                   "Technology".Substage := 116; //процесс прогрева
               ELSE
                   "HMI".INDICATION_TIME_1 := 255;
                   "HMI".INDICATION_TIME_2 := 255;
                   "Technology".Substage := 0; //неизвестно
           END_CASE;
       8:  //работа
           CASE "Technology".Regim_run_step OF
               0:
                   IF NOT "Protections_BLOCK".Not_flame_burner THEN
                       "HMI".LTIME_converter_IN := "Timer_RUN_temp_DB".ET;
                       "HMI".INDICATION_TIME_1 := DINT_TO_USINT("HMI".LTIME_converter_day);
                       "HMI".INDICATION_TIME_2 := INT_TO_USINT("HMI".LTIME_converter_hour);
                   ELSE    //если имеется блокировка защиты по погасанию пламени горелки
                       "HMI".TIME_converter_IN := "TON_protection_13_DB".PT - "TON_protection_13_DB".ET;
                       "HMI".INDICATION_TIME_1 := INT_TO_USINT("HMI".TIME_converter_minute);
                       "HMI".INDICATION_TIME_2 := INT_TO_USINT("HMI".TIME_converter_second);
                   END_IF;
                   "Technology".Substage := 117; //процесс работы 
               ELSE
                   "HMI".INDICATION_TIME_1 := 255;
                   "HMI".INDICATION_TIME_2 := 255;
                   "Technology".Substage := 0; //неизвестно
           END_CASE;
       9:  //экстренный останов
           "HMI".INDICATION_TIME_1 := 255;
           "HMI".INDICATION_TIME_2 := 255;
           CASE "Technology".Regim_emergency_stop_step OF
               0:
                   IF NOT "Message".EMERGENCY_STOP_not_initial_state THEN
                       "Technology".Substage := 120; //отключение всего 
                   ELSE
                       "Technology".Substage := 121; //устройства не переведены в исходное состояние
                   END_IF;
               ELSE
                   "Technology".Substage := 0; //неизвестно
           END_CASE;
       10: //аварийный останов
           "HMI".INDICATION_TIME_1 := 255;
           "HMI".INDICATION_TIME_2 := 255;
           CASE "Technology".Regim_alarm_stop_step OF
               0:
                   IF NOT "Message".ALARM_STOP_not_initial_state_gas THEN
                       "Technology".Substage := 122; //перевод всех газовых клапанов в исходное состояние
                   ELSE
                       "Technology".Substage := 123; //газовые клапана не переведены в исходное состояние
                   END_IF;
               ELSE
                   "Technology".Substage := 0; //неизвестно
           END_CASE;
       11: //плановый останов
           "HMI".INDICATION_TIME_1 := 255;
           "HMI".INDICATION_TIME_2 := 255;
           CASE "Technology".Regim_plan_stop_step OF
               0:
                   "Technology".Substage := 130; //вывод ЗРГ на значение минимальной мощности
               1:
                   "Technology".Substage := 131; //вывод ЗРГ на значение минимальной мощности
               2:
                   IF NOT "Message".PLAN_STOP_not_initial_state_gas THEN
                       "Technology".Substage := 132; //перевод газовых клапанов в исходное состояние, регуляторов разряжения и вентиляции на вентиляционные параметры
                   ELSE
                       "Technology".Substage := 133; //газовые клапана не переведены в исходное состояние
                   END_IF;
               3:
                   "Technology".Substage := 134; //перевод регуляторов разряжения и вентиляции на вентиляционные параметры
               ELSE
                   "Technology".Substage := 0; //неизвестно
           END_CASE;
       12: //постостановочная опрессовка
           "HMI".INDICATION_TIME_1 := 255;
           "HMI".INDICATION_TIME_2 := 255;
           CASE "Technology".Regim_stop_press_step OF
               0:
                   "Technology".Substage := 140; //анализ разрешения проведения постостановочной опрессовки
               1:
                   "Technology".Substage := 141; //контроль положения исполнительных механизмов по газу
               2:
                   "Technology".Substage := 142; //контроль min P
               3:
                   "Technology".Substage := 143; //контроль max P
               4:
                   "Technology".Substage := 144; //закрываем КБ
               5:
                   "Technology".Substage := 145; //контроль отсутствия давления газа м/у ПЗК
               6:
                   "Technology".Substage := 146; //открываем КО
               7:
                   "Technology".Substage := 147; //контроль достижения давления газа м/у ПЗК
               8:
                   "Technology".Substage := 148; //закрываем КО
               9:
                   "Technology".Substage := 149; //открываем КБ
               10:
                   "Technology".Substage := 150; //определение успешности постостановочной опрессовки
               11:
                   IF "Message".STOP_PRESS_PZK1_or_KO_untight THEN
                       "Technology".Substage := 151; //постостановочная опрессовка не прошла. ПЗК1 или КО негерметичен
                   END_IF;
                   IF "Message".STOP_PRESS_PZK2_or_KB_untight THEN
                       "Technology".Substage := 152; //постостановочная опрессовка не прошла. ПЗК2 или КБ негерметичен
                   END_IF;
                   IF "Message".STOP_PRESS_P_before_BG_min THEN
                       "Technology".Substage := 153; //постостановочная опрессовка не прошла. Низкое давление до БГ
                   END_IF;
                   IF "Message".STOP_PRESS_success THEN
                       "Technology".Substage := 154; //постостановочная опрессовка успешно проведена
                   END_IF;
               ELSE
                   "Technology".Substage := 0; //неизвестно
           END_CASE;
       13: //укороченная вентиляция
           CASE "Technology".Regim_short_ventilation_step OF
               0:
                   "HMI".INDICATION_TIME_1 := 255;
                   "HMI".INDICATION_TIME_2 := 255;
                   "Technology".Substage := 160; //анализ необходимости проведения укороченной вентиляции
               1:
                   "HMI".INDICATION_TIME_1 := 255;
                   "HMI".INDICATION_TIME_2 := 255;
                   "Technology".Substage := 161; //переход на поддержание вентиляционного значения разрежения
               2:
                   "HMI".INDICATION_TIME_1 := 255;
                   "HMI".INDICATION_TIME_2 := 255;
                   "Technology".Substage := 162; //переход на поддержание вентиляционного значения разрежения
               3:
                   "HMI".INDICATION_TIME_1 := 255;
                   "HMI".INDICATION_TIME_2 := 255;
                   "Technology".Substage := 163; //переход на поддержание вентиляционного значения давления воздуха
               4:
                   "HMI".TIME_converter_IN := "Timer_SHORT_VENTILATION_temp_DB".PT - "Timer_SHORT_VENTILATION_temp_DB".ET;
                   "HMI".INDICATION_TIME_1 := INT_TO_USINT("HMI".TIME_converter_minute);
                   "HMI".INDICATION_TIME_2 := INT_TO_USINT("HMI".TIME_converter_second);
                   "Technology".Substage := 164; //процесс вентиляции
               5:
                   "HMI".INDICATION_TIME_1 := 255;
                   "HMI".INDICATION_TIME_2 := 255;
                   "Technology".Substage := 165; //переход на поддержание розжигового значения разрежения
               6:
                   "HMI".INDICATION_TIME_1 := 255;
                   "HMI".INDICATION_TIME_2 := 255;
                   "Technology".Substage := 166; //переход на поддержание розжигового значения разрежения
               7:
                   "HMI".INDICATION_TIME_1 := 255;
                   "HMI".INDICATION_TIME_2 := 255;
                   "Technology".Substage := 167; //переход на поддержание розжигового значения давления воздуха
               ELSE
                   "HMI".INDICATION_TIME_1 := 255;
                   "HMI".INDICATION_TIME_2 := 255;
                   "Technology".Substage := 0; //неизвестно
           END_CASE;
       ELSE
           "Technology".Substage := 0; //неизвестно
   END_CASE;

   "TIME_converter_DB"(IN := "HMI".TIME_converter_IN,
                       Minute => "HMI".TIME_converter_minute,
                       Second => "HMI".TIME_converter_second);

   "LTIME_converter_DB"(IN := "HMI".LTIME_converter_IN,
                        Day=>"HMI".LTIME_converter_day,
                        Hour=>"HMI".LTIME_converter_hour);
END_FUNCTION

FUNCTION "Protection" : Void   // FC9, SCL
{ S7_Optimized_Access := 'TRUE' }
VERSION : 0.1
BEGIN
   (*Принудительный сброс блокировок защит*)
   (*Невоспламенение или погасание факела горелки котла*)
   "TON_protection_13_DB".TON(IN :="Protections_BLOCK".Not_flame_burner,
   PT := T#5m,
   Q => "Timer".protection_13_Q);
   IF "Timer".protection_13_Q THEN
       "Protections_BLOCK".Not_flame_burner := FALSE;
   END_IF;

   (*формирование обобщенного признака сработки защиты*)
   IF "Protections".P_gas_before_BG_max OR
       "Protections".P_gas_before_BG_min OR
       "Protections".P_gas_before_burner_min OR
       "Protections".P_gas_before_burner_max OR
       "Protections".DS_off OR
       "Protections".DV_off OR
       "Protections".dP_in_furnance_min OR
       "Protections".P_air_before_burner_min OR
       "Protections".L_water_min OR
       "Protections".L_water_max OR
       "Protections".P_steam_max OR
       "Protections".Not_flame_burner OR
       "Protections".Alarm_stop_HMI OR
       "Protections".Alarm_stop_SCADA THEN
       "Protections".Global := TRUE;
   ELSE
       "Protections".Global := FALSE;
   END_IF;
END_FUNCTION

FUNCTION "Regim_map" : Void   // FC10, SCL
{ S7_Optimized_Access := 'TRUE' }
VERSION : 0.1
BEGIN
   (*Защита от неправильного ввода параметров режимной карты*)
   IF "RegMap".P_gaz_2 < "RegMap".P_gaz_1 THEN
       "RegMap".P_gaz_2 := "RegMap".P_gaz_1+0.1;
   END_IF;
   IF "RegMap".P_gaz_3 < "RegMap".P_gaz_2 THEN
       "RegMap".P_gaz_3 := "RegMap".P_gaz_2+0.1;
   END_IF;
   IF "RegMap".P_gaz_4 < "RegMap".P_gaz_3 THEN
       "RegMap".P_gaz_4 := "RegMap".P_gaz_3+0.1;
   END_IF;
   IF "RegMap".P_gaz_5 < "RegMap".P_gaz_4 THEN
       "RegMap".P_gaz_5 := "RegMap".P_gaz_4+0.1;
   END_IF;
   IF "RegMap".P_gaz_6 < "RegMap".P_gaz_5 THEN
       "RegMap".P_gaz_6 := "RegMap".P_gaz_5+0.1;
   END_IF;
   IF "RegMap".P_gaz_7 < "RegMap".P_gaz_6 THEN
       "RegMap".P_gaz_7 := "RegMap".P_gaz_6+0.1;
   END_IF;
   IF "RegMap".P_gaz_8 < "RegMap".P_gaz_7 THEN
       "RegMap".P_gaz_8 := "RegMap".P_gaz_7+0.1;
   END_IF;

   (*НАСТРОЙКА РЕЖИМНОЙ КАРТЫ*)
   (*давление воздуха*)
   "Polyline_P_air_DB"();

   "Polyline_P_air_DB".Input := "P_gas_before_burner".Value;

   "Polyline_P_air_DB".UserData.Point[1].x := "RegMap".P_gaz_1;
   "Polyline_P_air_DB".UserData.Point[2].x := "RegMap".P_gaz_2;
   "Polyline_P_air_DB".UserData.Point[3].x := "RegMap".P_gaz_3;
   "Polyline_P_air_DB".UserData.Point[4].x := "RegMap".P_gaz_4;
   "Polyline_P_air_DB".UserData.Point[5].x := "RegMap".P_gaz_5;
   "Polyline_P_air_DB".UserData.Point[6].x := "RegMap".P_gaz_6;
   "Polyline_P_air_DB".UserData.Point[7].x := "RegMap".P_gaz_7;
   "Polyline_P_air_DB".UserData.Point[8].x := "RegMap".P_gaz_8;

   "Polyline_P_air_DB".UserData.Point[1].y := "RegMap".P_air_1;
   "Polyline_P_air_DB".UserData.Point[2].y := "RegMap".P_air_2;
   "Polyline_P_air_DB".UserData.Point[3].y := "RegMap".P_air_3;
   "Polyline_P_air_DB".UserData.Point[4].y := "RegMap".P_air_4;
   "Polyline_P_air_DB".UserData.Point[5].y := "RegMap".P_air_5;
   "Polyline_P_air_DB".UserData.Point[6].y := "RegMap".P_air_6;
   "Polyline_P_air_DB".UserData.Point[7].y := "RegMap".P_air_7;
   "Polyline_P_air_DB".UserData.Point[8].y := "RegMap".P_air_8;

   (*разряжение*)
   "Polyline_dP_DB"();

   "Polyline_dP_DB".Input := "P_gas_before_burner".Value;

   "Polyline_dP_DB".UserData.Point[1].x := "RegMap".P_gaz_1;
   "Polyline_dP_DB".UserData.Point[2].x := "RegMap".P_gaz_2;
   "Polyline_dP_DB".UserData.Point[3].x := "RegMap".P_gaz_3;
   "Polyline_dP_DB".UserData.Point[4].x := "RegMap".P_gaz_4;
   "Polyline_dP_DB".UserData.Point[5].x := "RegMap".P_gaz_5;
   "Polyline_dP_DB".UserData.Point[6].x := "RegMap".P_gaz_6;
   "Polyline_dP_DB".UserData.Point[7].x := "RegMap".P_gaz_7;
   "Polyline_dP_DB".UserData.Point[8].x := "RegMap".P_gaz_8;

   "Polyline_dP_DB".UserData.Point[1].y := "RegMap".dP_furnace_1;
   "Polyline_dP_DB".UserData.Point[2].y := "RegMap".dP_furnace_2;
   "Polyline_dP_DB".UserData.Point[3].y := "RegMap".dP_furnace_3;
   "Polyline_dP_DB".UserData.Point[4].y := "RegMap".dP_furnace_4;
   "Polyline_dP_DB".UserData.Point[5].y := "RegMap".dP_furnace_5;
   "Polyline_dP_DB".UserData.Point[6].y := "RegMap".dP_furnace_6;
   "Polyline_dP_DB".UserData.Point[7].y := "RegMap".dP_furnace_7;
   "Polyline_dP_DB".UserData.Point[8].y := "RegMap".dP_furnace_8;

   (*Режимная карта. Применить. Для журнала событий*)
   IF "RegMap".Apply THEN
       "HMI".RegMap_Apply_Log := TRUE;
   END_IF;

   IF "Syst".First_scan_reg_map THEN
       "RegMap".Apply := TRUE;
       "Syst".First_scan_reg_map := FALSE;
   END_IF;

   //применить новые значения
   "Polyline_P_air_DB".Validate := "RegMap".Apply;
   "Polyline_dP_DB".Validate := "RegMap".Apply;
   IF "RegMap".Apply THEN
       "RegMap".Apply := FALSE;
   END_IF;

   //значение расчетных параметров
   "RegMap".P_air_regim_map := "Polyline_P_air_DB".Output;
   "RegMap".dP_furnace_regim_map := "Polyline_dP_DB".Output;

   //индикация ошибки
   "RegMap".Error := "Polyline_P_air_DB".Error OR "Polyline_dP_DB".Error;

   //сброс
   "Polyline_P_air_DB".Reset := "RegMap".Reset;
   "Polyline_dP_DB".Reset := "RegMap".Reset;
   IF "RegMap".Reset THEN
       "RegMap".Reset := FALSE;
   END_IF;
END_FUNCTION

FUNCTION "Log" : Void   // FC11, SCL
{ S7_Optimized_Access := 'TRUE' }
VERSION : 0.1
BEGIN
   (*Нажатие кнопок для журнала событий*)
   (*Кнопка ВЕНТИЛЯЦИЯ на панели оператора для журнала событий*)
   IF "HMI".Btn_Ventilation_HMI THEN
       "HMI".Btn_Ventilation_HMI_Log := TRUE;
   END_IF;
   (*Кнопка ВЕНТИЛЯЦИЯ на SCADA для журнала событий*)
   IF "HMI".Btn_Ventilation_SCADA THEN
       "HMI".Btn_Ventilation_SCADA_Log := TRUE;
   END_IF;
   (*Кнопка ВЕНТИЛЯЦИЯ на ШАУ для журнала событий*)
   IF "Btn_Ventilation".Value THEN
       "HMI".Btn_Ventilation_ShAU_Log := TRUE;
   END_IF;
   (*Кнопка РОЗЖИГ на панели оператора для журнала событий*)
   IF "HMI".Btn_Ignition_HMI THEN
       "HMI".Btn_Ignition_HMI_Log := TRUE;
   END_IF;
   (*Кнопка РОЗЖИГ на SCADA для журнала событий*)
   IF "HMI".Btn_Ignition_SCADA THEN
       "HMI".Btn_Ignition_SCADA_Log := TRUE;
   END_IF;
   (*Кнопка РОЗЖИГ на ШАУ для журнала событий*)
   IF "Btn_Ignition".Value THEN
       "HMI".Btn_Ignition_ShAU_Log := TRUE;
   END_IF;
   (*Кнопка НОРМАЛЬНЫЙ ОСТАНОВ на панели оператора для журнала событий*)
   IF "HMI".Btn_normal_stop_HMI THEN
       "HMI".Btn_normal_stop_HMI_Log := TRUE;
   END_IF;
   (*Кнопка НОРМАЛЬНЫЙ ОСТАНОВ на SCADA для журнала событий*)
   IF "HMI".Btn_normal_stop_SCADA THEN
       "HMI".Btn_normal_stop_SCADA_Log := TRUE;
   END_IF;
   (*Кнопка АВАРИЙНЫЙ ОСТАНОВ на панели оператора для журнала событий*)
   IF "HMI".Btn_alarm_stop_HMI THEN
       "HMI".Btn_alarm_stop_HMI_Log := TRUE;
   END_IF;
   (*Кнопка АВАРИЙНЫЙ ОСТАНОВ на SCADA для журнала событий*)
   IF "HMI".Btn_alarm_stop_SCADA THEN
       "HMI".Btn_alarm_stop_SCADA_Log := TRUE;
   END_IF;
   (*Кнопка ЭКСТРЕННЫЙ ОСТАНОВ на ШАУ для журнала событий*)
   IF "Btn_STOP".Value THEN
       "HMI".Btn_emergency_stop_ShAU_Log := TRUE;
   END_IF;
   (*Кнопка ТЕСТОВАЯ ОПРЕССОВКА на панели оператора для журнала событий*)
   IF "HMI".Btn_test_press_HMI THEN
       "HMI".Btn_test_press_HMI_Log := TRUE;
   END_IF;
   (*Кнопка ТЕСТОВЫЙ РОЗЖИГ на панели оператора для журнала событий*)
   IF "HMI".Btn_test_ignition_HMI THEN
       "HMI".Btn_test_ignition_HMI_Log := TRUE;
   END_IF;
   (*Кнопка Ручной РОЗЖИГ на панели оператора для журнала событий*)
   IF "HMI".Btn_manual_ignition_HMI THEN
       "HMI".Btn_manual_ignition_HMI_Log := TRUE;
   END_IF;
   (*Кнопка СБРОС ЗВУКА на панели оператора для журнала событий*)
   IF "HMI".Btn_reset_sound_HMI THEN
       "HMI".Btn_reset_sound_HMI_Log := TRUE;
   END_IF;
   (*СБРОС аварий на ШАУ для журнала событий*)
   IF "Btn_Sound".Value THEN
       "HMI".Btn_reset_alarms_ShAU_Log := TRUE;
   END_IF;

   IF "HMI".Btn_Ventilation_HMI OR
       "HMI".Btn_Ventilation_SCADA OR
       "Btn_Ventilation".Value OR
       "HMI".Btn_Ignition_HMI OR
       "HMI".Btn_Ignition_SCADA OR
       "Btn_Ignition".Value OR
       "HMI".Btn_normal_stop_HMI OR
       "HMI".Btn_normal_stop_SCADA OR
       "HMI".Btn_alarm_stop_HMI OR
       "HMI".Btn_alarm_stop_SCADA OR
       "Btn_STOP".Value OR
       "HMI".Btn_test_press_HMI OR
       "HMI".Btn_test_ignition_HMI OR
       "HMI".Btn_manual_ignition_HMI OR
       "HMI".Btn_reset_sound_HMI OR
       "Alarm".Reset_alarms OR
       "Btn_Sound".Value OR
       "RegMap".Apply OR
       "Control_DS".Manual_Start OR
       "Control_DS".Manual_Stop OR
       "Control_DV".Manual_Start OR
       "Control_DV".Manual_Stop OR
       "Control_ZDG".Manual_open OR
       "Control_ZDG".Manual_close OR
       "Control_ZDG".Manual_stop OR
       "Control_GPZ".Manual_open OR
       "Control_GPZ".Manual_close OR
       "Control_GPZ".Manual_stop OR
       "Control_ZDSV_before_boiler".Manual_open OR
       "Control_ZDSV_before_boiler".Manual_close OR
       "Control_ZDSV_before_boiler".Manual_stop THEN
       "Timer".Log_IN := TRUE;
   END_IF;

   IF NOT "HMI".Btn_Ventilation_HMI AND
       NOT "HMI".Btn_Ventilation_SCADA AND
       NOT "Btn_Ventilation".Value AND
       NOT "HMI".Btn_Ignition_HMI AND
       NOT "HMI".Btn_Ignition_SCADA AND
       NOT "Btn_Ignition".Value AND
       NOT "HMI".Btn_normal_stop_HMI AND
       NOT "HMI".Btn_normal_stop_SCADA AND
       NOT "HMI".Btn_alarm_stop_HMI AND
       NOT "HMI".Btn_alarm_stop_SCADA AND
       NOT "Btn_STOP".Value AND
       NOT "HMI".Btn_test_press_HMI AND
       NOT "HMI".Btn_test_ignition_HMI AND
       NOT "HMI".Btn_manual_ignition_HMI AND
       NOT "HMI".Btn_reset_sound_HMI AND
       NOT "Alarm".Reset_alarms AND
       NOT "Btn_Sound".Value AND
       NOT "RegMap".Apply AND
       NOT "Control_DS".Manual_Start AND
       NOT "Control_DS".Manual_Stop AND
       NOT "Control_DV".Manual_Start AND
       NOT "Control_DV".Manual_Stop AND
       NOT "Control_ZDG".Manual_open AND
       NOT "Control_ZDG".Manual_close AND
       NOT "Control_ZDG".Manual_stop AND
       NOT "Control_GPZ".Manual_open AND
       NOT "Control_GPZ".Manual_close AND
       NOT "Control_GPZ".Manual_stop AND
       NOT "Control_ZDSV_before_boiler".Manual_open AND
       NOT "Control_ZDSV_before_boiler".Manual_close AND
       NOT "Control_ZDSV_before_boiler".Manual_stop THEN
       "Timer".Log_IN := FALSE;
   END_IF;

   "TOF_Log_DB".TOF(IN := "Timer".Log_IN,
   PT := "Timer".Log_PT,
   Q => "Timer".Log_Q);

   IF NOT "Timer".Log_Q THEN
       "HMI".Btn_Ventilation_HMI_Log := FALSE;
       "HMI".Btn_Ventilation_SCADA_Log := FALSE;
       "HMI".Btn_Ventilation_ShAU_Log := FALSE;
       "HMI".Btn_Ignition_HMI_Log := FALSE;
       "HMI".Btn_Ignition_SCADA_Log := FALSE;
       "HMI".Btn_Ignition_ShAU_Log := FALSE;
       "HMI".Btn_normal_stop_HMI_Log := FALSE;
       "HMI".Btn_normal_stop_SCADA_Log := FALSE;
       "HMI".Btn_alarm_stop_HMI_Log := FALSE;
       "HMI".Btn_alarm_stop_SCADA_Log := FALSE;
       "HMI".Btn_emergency_stop_ShAU_Log := FALSE;
       "HMI".Btn_test_press_HMI_Log := FALSE;
       "HMI".Btn_test_ignition_HMI_Log := FALSE;
       "HMI".Btn_manual_ignition_HMI_Log := FALSE;
       "HMI".Btn_reset_sound_HMI_Log := FALSE;
       "HMI".Reset_alarms_Log := FALSE;
       "HMI".Btn_reset_alarms_ShAU_Log := FALSE;
       "HMI".RegMap_Apply_Log := FALSE;
       "HMI".DS_Manual_Start_Log := FALSE;
       "HMI".DS_Manual_Stop_Log := FALSE;
       "HMI".DV_Manual_Start_Log := FALSE;
       "HMI".DV_Manual_Stop_Log := FALSE;
       "HMI".ZDG_Manual_open_Log := FALSE;
       "HMI".ZDG_Manual_close_Log := FALSE;
       "HMI".ZDG_Manual_stop_Log := FALSE;
       "HMI".GPZ_Manual_open_Log := FALSE;
       "HMI".GPZ_Manual_close_Log := FALSE;
       "HMI".GPZ_Manual_stop_Log := FALSE;
       "HMI".ZDSV_before_boiler_Manual_open_Log := FALSE;
       "HMI".ZDSV_before_boiler_Manual_close_Log := FALSE;
       "HMI".ZDSV_before_boiler_Manual_stop_Log := FALSE;
   END_IF;
END_FUNCTION

FUNCTION "Select_regim" : Void   // FC12, SCL
{ S7_Optimized_Access := 'TRUE' }
VERSION : 0.1
BEGIN
   (*Выбор режима работы*)
   (*  1-ОТКЛ
       2-ПРОВЕРКА
       3-ВЕНТИЛЯЦИЯ
       4-ОПРЕССОВКА
       5-РОЗЖИГ
       6-ВЫХОД НА МИНИМАЛЬНУЮ МОЩНОСТЬ
       7-ПРОГРЕВ
       8-РАБОТА
       9-ЭКСТРЕННЫЙ ОСТАНОВ
       10-АВАРИЙНЫЙ ОСТАНОВ
       11-ПЛАНОВЫЙ ОСТАНОВ
       12-ПОСТОСТАНОВОЧНАЯ ОПРЕССОВКА
       13-УКОРОЧЕННАЯ ВЕНТИЛЯЦИЯ*)
   IF "Technology".Regim <= 0 OR "Technology".Regim >= 16 THEN
       "Technology".Regim := 1;
   END_IF;

   (*Экстренный останов*)
   IF "Btn_STOP".Value THEN
       "Technology".Regim := 9;
   END_IF;

   (*Аварийный останов*)
   IF "Protections".Global THEN
       "Technology".Regim := 10;
   END_IF;

   (*Плановый останов*)
   IF ("FRONT".Btn_Normal_stop_HMI OR "FRONT".Btn_Normal_stop_SCADA) AND "Technology".Regim <> 1 AND
       "Technology".Regim <> 10 AND
       "Technology".Regim <> 12 THEN
       "Technology".Regim := 11;
   END_IF;

   (*сброс признака провентилированности топки*)
   IF "PZK2_not_close".Value OR
       ((NOT "DS_invertor_on".Value AND NOT "DS_powergrid_on".Value) OR (NOT "DV_invertor_on".Value AND NOT "DV_powergrid_on".Value)) THEN
       "Technology".Ventilation_conducted := FALSE;
   END_IF;

   (*был переход в режим РОЗЖИГ и открытие ПЗК2*)
   IF "Technology".Ventilation_conducted THEN
       "Technology".transition_ignition := FALSE;
   END_IF;
   IF "Technology".Regim = 5 AND "PZK2_not_close".Value THEN
       "Technology".transition_ignition := TRUE;
   END_IF;

   (*если текущий режим не ОТКЛ и не РУЧНОЙ РОЗЖИГ, то ИМ по газу принудительно переводим в автоматический режим *)
   IF "Technology".Regim = 1 OR
       ("Technology".Regim = 5 AND "Technology".Regim_ignition_step =19) THEN
       ;
   ELSE
       (*КБ*)
       "Control_KB".Mode := TRUE;
       (*KO*)
       "Control_KO".Mode := TRUE;
       (*КЗ*)
       "Control_KZ".Mode := TRUE;
       (*ПЗК1*)
       "Control_PZK1".Mode := TRUE;
       (*ПЗК2*)
       "Control_PZK2".Mode := TRUE;
       (*ЗДГ*)
       //"Control_ZDG".Mode := TRUE;
       (*ИВН*)
       "Control_IVN".Mode := TRUE;
   END_IF;

   (*сброс признака тестовой опрессовки, если текущий режим не вентиляция и не опрессовка*)
   IF "Technology".Regim <> 3 AND "Technology".Regim <> 4 THEN
       "Technology".Test_press_run := FALSE;
       "Message".TEST_PRESS_ok := FALSE;   //сброс сообщения об успешном прохождении тестовой опрессовки
   END_IF;

   (*Взведение и снятие защит нажатию кнопок аварийного останова*)
   IF "Technology".Regim = 2 OR
       "Technology".Regim = 3 OR
       "Technology".Regim = 4 OR
       "Technology".Regim = 5 OR
       "Technology".Regim = 6 OR
       "Technology".Regim = 7 OR
       "Technology".Regim = 8 OR
       "Technology".Regim = 11 THEN
       //взводим защиту Нажата кнопка аварийного останова на панели оператора
       "Alarm_Enable".Alarm_stop_HMI := TRUE;
       //взводим защиту Нажата кнопка аварийного останова на SCADA
       "Alarm_Enable".Alarm_stop_SCADA := TRUE;
   ELSE
       //снимаем защиту Нажата кнопка аварийного останова на панели оператора
       "Alarm_Enable".Alarm_stop_HMI := FALSE;
       //снимаем защиту Нажата кнопка аварийного останова на SCADA
       "Alarm_Enable".Alarm_stop_SCADA := FALSE;
   END_IF;

   (*Аварийные сообщения по загазованности (не являются защитами)*)
   //СО2 порог 2
   "Alarm_Enable".CO2 := TRUE;
   //CH4
   "Alarm_Enable".CH4 := TRUE;

   IF "Technology".SP_L_water < -300.0 THEN
       "Technology".SP_L_water := -300.0;
   END_IF;
   IF "Technology".SP_L_water > 300.0 THEN
       "Technology".SP_L_water := 300.0;
   END_IF;

   IF "Technology".SP_P_steam < 0.0 THEN
       "Technology".SP_P_steam := 0.0;
   END_IF;
   IF "Technology".SP_P_steam > "P_steam".HL_sensor THEN
       "Technology".SP_P_steam := "P_steam".HL_sensor;
   END_IF;
END_FUNCTION

FUNCTION "Indication" : Void   // FC15, SCL
{ S7_Optimized_Access := 'TRUE' }
VERSION : 0.1
BEGIN
   (*Управление индикацией*)
   //генератор импульсов
   "Timer_IND_1_DB".TON(IN := "Timer".IND_1_IN,
                        PT := "Timer".IND_1_PT,
                        Q => "Timer".IND_1_Q);
   "Timer_IND_2_DB".TON(IN := "Timer".IND_2_IN,
                        PT := "Timer".IND_2_PT,
                        Q => "Timer".IND_2_Q);
   "Timer".IND_1_PT := T#1s;
   "Timer".IND_2_PT := T#1s;
   IF NOT "Timer".IND_1_IN AND NOT "Timer".IND_2_IN THEN
       "Timer".IND_1_IN := TRUE;
   END_IF;
   IF "Timer".IND_1_Q THEN
       "Timer".IND_1_IN := FALSE;
       "Timer".IND_2_IN := TRUE;
       "Syst".Gen_imp := FALSE;
   END_IF;
   IF "Timer".IND_2_Q THEN
       "Timer".IND_2_IN := FALSE;
       "Timer".IND_1_IN := TRUE;
       "Syst".Gen_imp := TRUE;
   END_IF;

   (*Индикация «Работа»*)
   IF "Technology".Regim <> 5 AND
       "Technology".Regim <> 6 AND
       "Technology".Regim <> 7 AND
       "Technology".Regim <> 8 THEN
       "Indication_RUN".Value := FALSE;
   END_IF;
   IF "Technology".Regim = 5 OR
       "Technology".Regim = 6 OR
       "Technology".Regim = 7 THEN
       "Indication_RUN".Value := "Syst".Gen_imp;
   END_IF;
   IF "Technology".Regim = 8 THEN
       "Indication_RUN".Value := TRUE;
   END_IF;

   (*Индикация «Авария»*)
   IF "Alarm".P_gas_before_BG_max OR
       "Alarm".P_gas_before_BG_min OR
       "Alarm".P_gas_before_burner_min OR
       "Alarm".P_gas_before_burner_max OR
       "Alarm".DS_off OR
       "Alarm".DV_off OR
       "Alarm".dP_furnace_boiler_min OR
       "Alarm".P_air_before_burner_min OR
       "Alarm".L_water_min OR
       "Alarm".L_water_max OR
       "Alarm".P_steam_max OR
       "Alarm".Not_flame_burner OR
       "Alarm".Alarm_stop_HMI OR
       "Alarm".Alarm_stop_SCADA OR
       "Alarm".CO2 OR
       "Alarm".CH4 THEN
       "Indication_ALARM".Value := TRUE;
   ELSE
       IF "TON_alarm_1_DB".IN OR
           "TON_alarm_2_DB".IN OR
           "TON_alarm_3_DB".IN OR
           "TON_alarm_4_DB".IN OR
           "TON_alarm_5_DB".IN OR
           "TON_alarm_6_DB".IN OR
           "TON_alarm_7_DB".IN OR
           "TON_alarm_8_DB".IN OR
           "TON_alarm_9_DB".IN OR
           "TON_alarm_10_DB".IN OR
           "TON_alarm_11_DB".IN OR
           "TON_alarm_12_DB".IN OR
           "TON_alarm_13_DB".IN OR
           "TON_alarm_14_DB".IN OR
           "TON_alarm_15_DB".IN OR
           "TON_alarm_16_DB".IN OR
           "FRONT".Btn_Alarm_stop_HMI OR
           "FRONT".Btn_Alarm_stop_SCADA THEN
           "Indication_ALARM".Value := "Syst".Gen_imp;
       ELSE
           "Indication_ALARM".Value := FALSE;
       END_IF;
   END_IF;

   (*Индикация «Защиты в норме»*)
   IF "Protections".Global THEN
       "Indication_NORMA".Value := FALSE;
   ELSE
       IF "Protections_BLOCK".P_gas_before_BG_max OR
           "Protections_BLOCK".P_gas_before_BG_min OR
           "Protections_BLOCK".P_gas_before_burner_min OR
           "Protections_BLOCK".P_gas_before_burner_max OR
           "Protections_BLOCK".DS_off OR
           "Protections_BLOCK".DV_off OR
           "Protections_BLOCK".dP_in_furnance_min OR
           "Protections_BLOCK".P_air_before_burner_min OR
           "Protections_BLOCK".L_water_min OR
           "Protections_BLOCK".L_water_max OR
           "Protections_BLOCK".P_steam_max OR
           "Protections_BLOCK".Not_flame_burner OR
           "Protections_BLOCK".Alarm_stop_HMI OR
           "Protections_BLOCK".Alarm_stop_SCADA THEN
           "Indication_NORMA".Value := "Syst".Gen_imp;
       ELSE
           "Indication_NORMA".Value := TRUE;
       END_IF;
   END_IF;

   (*Индикация «Готов к розжигу»*)
   IF "Technology".Regim = 3 AND "Technology".Regim_ventilation_step = 25 THEN
       "Indication_READY".Value := "Syst".Gen_imp;
   ELSE
       "Indication_READY".Value := FALSE;
   END_IF;
END_FUNCTION

FUNCTION "Control_Device" : Void   // FC25, SCL
{ S7_Optimized_Access := 'TRUE' }
VERSION : 0.1
BEGIN
   (*ДС. Ручное управление. Пуск. Для журнала событий*)
   IF "Control_DS".Manual_Start THEN
       "HMI".DS_Manual_Start_Log := TRUE;
   END_IF;
   (*ДС. Ручное управление. Стоп. Для журнала событий*)
   IF "Control_DS".Manual_Stop THEN
       "HMI".DS_Manual_Stop_Log := TRUE;
   END_IF;
   (*ДВ. Ручное управление. Пуск. Для журнала событий*)
   IF "Control_DV".Manual_Start THEN
       "HMI".DV_Manual_Start_Log := TRUE;
   END_IF;
   (*ДВ. Ручное управление. Стоп. Для журнала событий*)
   IF "Control_DV".Manual_Stop THEN
       "HMI".DV_Manual_Stop_Log := TRUE;
   END_IF;
   (*ЗДГ. Ручное управление. Открыть. Для журнала событий*)
   IF "Control_ZDG".Manual_open THEN
       "HMI".ZDG_Manual_open_Log := TRUE;
   END_IF;
   (*ЗДГ. Ручное управление. Закрыть. Для журнала событий*)
   IF "Control_ZDG".Manual_close THEN
       "HMI".ZDG_Manual_close_Log := TRUE;
   END_IF;
   (*ЗДГ. Ручное управление. Стоп. Для журнала событий*)
   IF "Control_ZDG".Manual_stop THEN
       "HMI".ZDG_Manual_stop_Log := TRUE;
   END_IF;
   (*ГПЗ. Ручное управление. Открыть. Для журнала событий*)
   IF "Control_GPZ".Manual_open THEN
       "HMI".GPZ_Manual_open_Log := TRUE;
   END_IF;
   (*ГПЗ. Ручное управление. Закрыть. Для журнала событий*)
   IF "Control_GPZ".Manual_close THEN
       "HMI".GPZ_Manual_close_Log := TRUE;
   END_IF;
   (*ГПЗ. Ручное управление. Стоп. Для журнала событий*)
   IF "Control_GPZ".Manual_stop THEN
       "HMI".GPZ_Manual_stop_Log := TRUE;
   END_IF;
   (*ЗДСВ перед котлом. Ручное управление. Открыть. Для журнала событий*)
   IF "Control_ZDSV_before_boiler".Manual_open THEN
       "HMI".ZDSV_before_boiler_Manual_open_Log := TRUE;
   END_IF;
   (*ЗДСВ перед котлом. Ручное управление. Закрыть. Для журнала событий*)
   IF "Control_ZDSV_before_boiler".Manual_close THEN
       "HMI".ZDSV_before_boiler_Manual_close_Log := TRUE;
   END_IF;
   (*ЗДСВ перед котлом. Ручное управление. Стоп. Для журнала событий*)
   IF "Control_ZDSV_before_boiler".Manual_stop THEN
       "HMI".ZDSV_before_boiler_Manual_stop_Log := TRUE;
   END_IF;

   (*Управление исполнительными механизмами*)
   (*ЗРГ*)
   //проверка и сброс ручных команд
   //сброс обеих команд при автоматическом режиме
   IF "Control_ZRG".Mode THEN
       "Control_ZRG".Manual_open := FALSE;
       "Control_ZRG".Manual_close := FALSE;
   END_IF;
   //сброс обеих команд при их одновременном наличии
   IF "Control_ZRG".Manual_open AND "Control_ZRG".Manual_close THEN
       "Control_ZRG".Manual_open := FALSE;
       "Control_ZRG".Manual_close := FALSE;
   END_IF;
   //сброс ручной команды на открытие при полном открытии
   IF "ZRG_open".Value THEN
       "Control_ZRG".Manual_open := FALSE;
   END_IF;
   //сброс ручной команды на закрытие при полном закрытии
   IF "ZRG_close".Value THEN
       "Control_ZRG".Manual_close := FALSE;
   END_IF;
   //проверка и сброс ручных команд от ПЛК
   //сброс обеих команд при режиме полного автомата
   IF "Control_ZRG".Mode_from_PLC THEN
       "Control_ZRG".Manual_open_from_PLC := FALSE;
       "Control_ZRG".Manual_close_from_PLC := FALSE;
   END_IF;
   //сброс обеих команд от ПЛК при их одновременном наличии
   IF "Control_ZRG".Manual_open_from_PLC AND "Control_ZRG".Manual_close_from_PLC THEN
       "Control_ZRG".Manual_open_from_PLC := FALSE;
       "Control_ZRG".Manual_close_from_PLC := FALSE;
   END_IF;
   //сброс ручной команды на открытие от ПЛК при полном открытии
   IF "ZRG_open".Value THEN
       "Control_ZRG".Manual_open_from_PLC := FALSE;
   END_IF;
   //сброс ручной команды на закрытие от ПЛК при полном закрытии
   IF "ZRG_close".Value THEN
       "Control_ZRG".Manual_close_from_PLC := FALSE;
   END_IF;
   //управление
   IF "ZRG_avto".Value THEN
       IF "Technology".Regim <> 11 THEN
           "Control_ZRG".SP_PID := "Technology".SP_P_steam;
       END_IF;
       IF ("Control_ZRG".Mode AND "Control_ZRG".Mode_from_PLC AND NOT "P_steam".Error_sensor) THEN //автоматический режим
           "PID_impulse_ZRG_DB"(DIR := TRUE,
                                PV := "P_steam".Value,
                                SP := "Control_ZRG".SP_PID,
                                DB := "Control_ZRG".DB_PID,
                                KP := "Control_ZRG".KP_PID,
                                TI := "Control_ZRG".TI_PID,
                                TD := "Control_ZRG".TD_PID,
                                CYCLE := 100,
                                FMT := "Control_ZRG".FMT_PID,
                                DT_MIN := "Control_ZRG".DT_MIN_PID,
                                AUTO := ("Control_ZRG".Mode AND "Control_ZRG".Mode_from_PLC AND NOT "P_steam".Error_sensor),
                                MORE := ((NOT "Control_ZRG".Mode AND "Control_ZRG".Manual_open) OR ("Control_ZRG".Mode AND "Control_ZRG".Manual_open_from_PLC)),
                                LESS := ((NOT "Control_ZRG".Mode AND "Control_ZRG".Manual_close) OR ("Control_ZRG".Mode AND "Control_ZRG".Manual_close_from_PLC)),
                                Hold := false,
                                GAP := "Control_ZRG".GAP,
                                PLUS := "ZRG_control_open".Value,
                                MINUS := "ZRG_control_close".Value);
       ELSE //ручной режим
           "PID_impulse_ZRG_DB"(DIR := TRUE,
                                PV := "P_steam".Value,
                                SP := "P_steam".Value,
                                DB := "Control_ZRG".DB_PID,
                                KP := "Control_ZRG".KP_PID,
                                TI := "Control_ZRG".TI_PID,
                                TD := "Control_ZRG".TD_PID,
                                CYCLE := 100,
                                FMT := "Control_ZRG".FMT_PID,
                                DT_MIN := "Control_ZRG".DT_MIN_PID,
                                AUTO := ("Control_ZRG".Mode AND "Control_ZRG".Mode_from_PLC AND NOT "P_steam".Error_sensor),
                                MORE := ((NOT "Control_ZRG".Mode AND "Control_ZRG".Manual_open) OR ("Control_ZRG".Mode AND "Control_ZRG".Manual_open_from_PLC)),
                                LESS := ((NOT "Control_ZRG".Mode AND "Control_ZRG".Manual_close) OR ("Control_ZRG".Mode AND "Control_ZRG".Manual_close_from_PLC)),
                                Hold := false,
                                GAP := "Control_ZRG".GAP,
                                PLUS := "ZRG_control_open".Value,
                                MINUS := "ZRG_control_close".Value);
       END_IF;
   ELSE
       //при переводе БРУ в ручной режим
       "ZRG_control_open".Value := FALSE;
       "ZRG_control_close".Value := FALSE;
       "Control_ZRG".Manual_open := FALSE;
       "Control_ZRG".Manual_close := FALSE;
       "PID_impulse_ZRG_DB"(DIR := TRUE,
                            PV := "P_steam".Value,
                            SP := "P_steam".Value,
                            DB := "Control_ZRG".DB_PID,
                            KP := "Control_ZRG".KP_PID,
                            TI := "Control_ZRG".TI_PID,
                            TD := "Control_ZRG".TD_PID,
                            CYCLE := 100,
                            FMT := "Control_ZRG".FMT_PID,
                            DT_MIN := "Control_ZRG".DT_MIN_PID,
                            AUTO := FALSE,
                            MORE := FALSE,
                            LESS := FALSE,
                            Hold := false,
                            GAP := "Control_ZRG".GAP,
                            PLUS := "ZRG_control_open".Value,
                            MINUS := "ZRG_control_close".Value);
   END_IF;
   //ораничение на открытие по max давлению газа в режиме ПРОГРЕВ
   IF "Technology".Regim = 7 AND "P_gas_before_burner".Value > "Technology".Max_P_gas_heating THEN
       "ZRG_control_open".Value := FALSE;
   END_IF;
   //ораничение на открытие по давлению газа из режимной карты в режиме РАБОТА
   IF "Technology".Regim = 8 AND "P_gas_before_burner".Value > "RegMap".P_gaz_8 THEN
       "ZRG_control_open".Value := FALSE;
   END_IF;
   //ограничение по закрытию ниже режима min мощности в режиме ПРОГРЕВ и РАБОТА
   IF ("Technology".Regim = 7 OR "Technology".Regim = 8) AND NOT "ZRG_middle".Value THEN
       "ZRG_control_close".Value := FALSE;
   END_IF;

   (*ЗРВ*)
   //проверка и сброс ручных команд
   //сброс обеих команд при автоматическом режиме
   IF "Control_ZRW".Mode THEN
       "Control_ZRW".Manual_open := FALSE;
       "Control_ZRW".Manual_close := FALSE;
   END_IF;
   //сброс обеих команд при их одновременном наличии
   IF "Control_ZRW".Manual_open AND "Control_ZRW".Manual_close THEN
       "Control_ZRW".Manual_open := FALSE;
       "Control_ZRW".Manual_close := FALSE;
   END_IF;
   //сброс ручной команды на открытие при полном открытии
   IF "ZRW_open".Value THEN
       "Control_ZRW".Manual_open := FALSE;
   END_IF;
   //сброс ручной команды на закрытие при полном закрытии
   IF "ZRW_close".Value THEN
       "Control_ZRW".Manual_close := FALSE;
   END_IF;
   //проверка и сброс ручных команд от ПЛК
   //сброс обеих команд при режиме полного автомата
   IF "Control_ZRW".Mode_from_PLC THEN
       "Control_ZRW".Manual_open_from_PLC := FALSE;
       "Control_ZRW".Manual_close_from_PLC := FALSE;
   END_IF;
   //сброс обеих команд от ПЛК при их одновременном наличии
   IF "Control_ZRW".Manual_open_from_PLC AND "Control_ZRW".Manual_close_from_PLC THEN
       "Control_ZRW".Manual_open_from_PLC := FALSE;
       "Control_ZRW".Manual_close_from_PLC := FALSE;
   END_IF;
   //сброс ручной команды на открытие от ПЛК при полном открытии
   IF "ZRW_open".Value THEN
       "Control_ZRW".Manual_open_from_PLC := FALSE;
   END_IF;
   //сброс ручной команды на закрытие от ПЛК при полном закрытии
   IF "ZRW_close".Value THEN
       "Control_ZRW".Manual_close_from_PLC := FALSE;
   END_IF;
   //управление
   IF "ZRW_avto".Value THEN
       "Control_ZRW".SP_PID := "Technology".SP_L_water;
       IF ("Control_ZRW".Mode AND "Control_ZRW".Mode_from_PLC AND NOT "L_water".Error_sensor) THEN //автоматический режим
           "PID_impulse_ZRW_DB"(DIR := TRUE,
                                PV := "L_water".Value,
                                SP := "Control_ZRW".SP_PID,
                                DB := "Control_ZRW".DB_PID,
                                KP := "Control_ZRW".KP_PID,
                                TI := "Control_ZRW".TI_PID,
                                TD := "Control_ZRW".TD_PID,
                                CYCLE := 100,
                                FMT := "Control_ZRW".FMT_PID,
                                DT_MIN := "Control_ZRW".DT_MIN_PID,
                                AUTO := ("Control_ZRW".Mode AND "Control_ZRW".Mode_from_PLC AND NOT "L_water".Error_sensor),
                                MORE := ((NOT "Control_ZRW".Mode AND "Control_ZRW".Manual_open) OR ("Control_ZRW".Mode AND "Control_ZRW".Manual_open_from_PLC)),
                                LESS := ((NOT "Control_ZRW".Mode AND "Control_ZRW".Manual_close) OR ("Control_ZRW".Mode AND "Control_ZRW".Manual_close_from_PLC)),
                                Hold := false,
                                GAP := "Control_ZRW".GAP,
                                PLUS := "ZRW_control_open".Value,
                                MINUS := "ZRW_control_close".Value);
       ELSE    //ручной режим
           "PID_impulse_ZRW_DB"(DIR := TRUE,
                                PV := "L_water".Value,
                                SP := "L_water".Value,
                                DB := "Control_ZRW".DB_PID,
                                KP := "Control_ZRW".KP_PID,
                                TI := "Control_ZRW".TI_PID,
                                TD := "Control_ZRW".TD_PID,
                                CYCLE := 100,
                                FMT := "Control_ZRW".FMT_PID,
                                DT_MIN := "Control_ZRW".DT_MIN_PID,
                                AUTO := ("Control_ZRW".Mode AND "Control_ZRW".Mode_from_PLC AND NOT "L_water".Error_sensor),
                                MORE := ((NOT "Control_ZRW".Mode AND "Control_ZRW".Manual_open) OR ("Control_ZRW".Mode AND "Control_ZRW".Manual_open_from_PLC)),
                                LESS := ((NOT "Control_ZRW".Mode AND "Control_ZRW".Manual_close) OR ("Control_ZRW".Mode AND "Control_ZRW".Manual_close_from_PLC)),
                                Hold := false,
                                GAP := "Control_ZRW".GAP,
                                PLUS := "ZRW_control_open".Value,
                                MINUS := "ZRW_control_close".Value);
       END_IF;
   ELSE
       //при переводе БРУ в ручной режим
       "ZRW_control_open".Value := FALSE;
       "ZRW_control_close".Value := FALSE;
       "Control_ZRW".Manual_open := FALSE;
       "Control_ZRW".Manual_close := FALSE;
       "PID_impulse_ZRW_DB"(DIR := TRUE,
                            PV := "L_water".Value,
                            SP := "L_water".Value,
                            DB := "Control_ZRW".DB_PID,
                            KP := "Control_ZRW".KP_PID,
                            TI := "Control_ZRW".TI_PID,
                            TD := "Control_ZRW".TD_PID,
                            CYCLE := 100,
                            FMT := "Control_ZRW".FMT_PID,
                            DT_MIN := "Control_ZRW".DT_MIN_PID,
                            AUTO := FALSE,
                            MORE := FALSE,
                            LESS := FALSE,
                            Hold := false,
                            GAP := "Control_ZRW".GAP,
                            PLUS := "ZRW_control_open".Value,
                            MINUS := "ZRW_control_close".Value);
   END_IF;

   (*НАВ*)
   //проверка и сброс ручных команд
   //сброс обеих команд при автоматическом режиме
   IF "Control_NAV".Mode THEN
       "Control_NAV".Manual_open := FALSE;
       "Control_NAV".Manual_close := FALSE;
   END_IF;
   //сброс обеих команд при их одновременном наличии
   IF "Control_NAV".Manual_open AND "Control_NAV".Manual_close THEN
       "Control_NAV".Manual_open := FALSE;
       "Control_NAV".Manual_close := FALSE;
   END_IF;
   //сброс ручной команды на открытие при полном открытии
   IF "NAV_open".Value THEN
       "Control_NAV".Manual_open := FALSE;
   END_IF;
   //сброс ручной команды на закрытие при полном закрытии
   IF "NAV_close".Value THEN
       "Control_NAV".Manual_close := FALSE;
   END_IF;
   //проверка и сброс ручных команд от ПЛК
   //сброс обеих команд при режиме полного автомата
   IF "Control_NAV".Mode AND "Control_NAV".Mode_from_PLC THEN
       "Control_NAV".Manual_open_from_PLC := FALSE;
       "Control_NAV".Manual_close_from_PLC := FALSE;
   END_IF;
   //сброс обеих команд от ПЛК при их одновременном наличии
   IF "Control_NAV".Manual_open_from_PLC AND "Control_NAV".Manual_close_from_PLC THEN
       "Control_NAV".Manual_open_from_PLC := FALSE;
       "Control_NAV".Manual_close_from_PLC := FALSE;
   END_IF;
   //сброс ручной команды на открытие от ПЛК при полном открытии
   IF "NAV_open".Value THEN
       "Control_NAV".Manual_open_from_PLC := FALSE;
   END_IF;
   //сброс ручной команды на закрытие от ПЛК при полном закрытии
   IF "NAV_close".Value THEN
       "Control_NAV".Manual_close_from_PLC := FALSE;
   END_IF;
   //управление
   IF "NAV_avto".Value THEN
       IF ("Control_NAV".Mode AND "Control_NAV".Mode_from_PLC AND NOT "P_air_burner".Error_sensor) THEN //автоматический режим
           "PID_impulse_NAV_DB"(DIR := TRUE,
                                PV := "P_air_burner".Value,
                                SP := "Control_NAV".SP_PID,
                                DB := "Control_NAV".DB_PID,
                                KP := "Control_NAV".KP_PID,
                                TI := "Control_NAV".TI_PID,
                                TD := "Control_NAV".TD_PID,
                                CYCLE := 100,
                                FMT := "Control_NAV".FMT_PID,
                                DT_MIN := "Control_NAV".DT_MIN_PID,
                                AUTO := ("Control_NAV".Mode AND "Control_NAV".Mode_from_PLC AND NOT "P_air_burner".Error_sensor),
                                MORE := ((NOT "Control_NAV".Mode AND "Control_NAV".Manual_open) OR ("Control_NAV".Mode AND "Control_NAV".Manual_open_from_PLC)),
                                LESS := ((NOT "Control_NAV".Mode AND "Control_NAV".Manual_close) OR ("Control_NAV".Mode AND "Control_NAV".Manual_close_from_PLC)),
                                Hold := false,
                                GAP := "Control_NAV".GAP,
                                PLUS := "NAV_control_open".Value,
                                MINUS := "NAV_control_close".Value);
       ELSE    //ручной режим
           "PID_impulse_NAV_DB"(DIR := TRUE,
                                PV := "P_air_burner".Value,
                                SP := "P_air_burner".Value,
                                DB := "Control_NAV".DB_PID,
                                KP := "Control_NAV".KP_PID,
                                TI := "Control_NAV".TI_PID,
                                TD := "Control_NAV".TD_PID,
                                CYCLE := 100,
                                FMT := "Control_NAV".FMT_PID,
                                DT_MIN := "Control_NAV".DT_MIN_PID,
                                AUTO := ("Control_NAV".Mode AND "Control_NAV".Mode_from_PLC AND NOT "P_air_burner".Error_sensor),
                                MORE := ((NOT "Control_NAV".Mode AND "Control_NAV".Manual_open) OR ("Control_NAV".Mode AND "Control_NAV".Manual_open_from_PLC)),
                                LESS := ((NOT "Control_NAV".Mode AND "Control_NAV".Manual_close) OR ("Control_NAV".Mode AND "Control_NAV".Manual_close_from_PLC)),
                                Hold := false,
                                GAP := "Control_NAV".GAP,
                                PLUS := "NAV_control_open".Value,
                                MINUS := "NAV_control_close".Value);
       END_IF;
   ELSE
       //при переводе БРУ в ручной режим
       "NAV_control_open".Value := FALSE;
       "NAV_control_close".Value := FALSE;
       "Control_NAV".Manual_open := FALSE;
       "Control_NAV".Manual_close := FALSE;
       "PID_impulse_NAV_DB"(DIR := TRUE,
                            PV := "P_air_burner".Value,
                            SP := "P_air_burner".Value,
                            DB := "Control_NAV".DB_PID,
                            KP := "Control_NAV".KP_PID,
                            TI := "Control_NAV".TI_PID,
                            TD := "Control_NAV".TD_PID,
                            CYCLE := 100,
                            FMT := "Control_NAV".FMT_PID,
                            DT_MIN := "Control_NAV".DT_MIN_PID,
                            AUTO := FALSE,
                            MORE := FALSE,
                            LESS := FALSE,
                            Hold := false,
                            GAP := "Control_NAV".GAP,
                            PLUS := "NAV_control_open".Value,
                            MINUS := "NAV_control_close".Value);
   END_IF;

   (*НАД*)
   //проверка и сброс ручных команд
   //сброс обеих команд при автоматическом режиме
   IF "Control_NAD".Mode THEN
       "Control_NAD".Manual_open := FALSE;
       "Control_NAD".Manual_close := FALSE;
   END_IF;
   //сброс обеих команд при их одновременном наличии
   IF "Control_NAD".Manual_open AND "Control_NAD".Manual_close THEN
       "Control_NAD".Manual_open := FALSE;
       "Control_NAD".Manual_close := FALSE;
   END_IF;
   //сброс ручной команды на открытие при полном открытии
   IF "NAD_open".Value THEN
       "Control_NAD".Manual_open := FALSE;
   END_IF;
   //сброс ручной команды на закрытие при полном закрытии
   IF "NAD_close".Value THEN
       "Control_NAD".Manual_close := FALSE;
   END_IF;
   //проверка и сброс ручных команд от ПЛК
   //сброс обеих команд при режиме полного автомата
   IF "Control_NAD".Mode AND "Control_NAD".Mode_from_PLC THEN
       "Control_NAD".Manual_open_from_PLC := FALSE;
       "Control_NAD".Manual_close_from_PLC := FALSE;
   END_IF;
   //сброс обеих команд от ПЛК при их одновременном наличии
   IF "Control_NAD".Manual_open_from_PLC AND "Control_NAD".Manual_close_from_PLC THEN
       "Control_NAD".Manual_open_from_PLC := FALSE;
       "Control_NAD".Manual_close_from_PLC := FALSE;
   END_IF;
   //сброс ручной команды на открытие от ПЛК при полном открытии
   IF "NAD_open".Value THEN
       "Control_NAD".Manual_open_from_PLC := FALSE;
   END_IF;
   //сброс ручной команды на закрытие от ПЛК при полном закрытии
   IF "NAD_close".Value THEN
       "Control_NAD".Manual_close_from_PLC := FALSE;
   END_IF;
   //управление
   IF "NAD_avto".Value THEN
       IF ("Control_NAD".Mode AND "Control_NAD".Mode_from_PLC AND NOT "dP_furnace_boiler".Error_sensor) THEN   //автоматический режим
           "PID_impulse_NAD_DB"(DIR := FALSE,
                                PV := "dP_furnace_boiler".Value,
                                SP := "Control_NAD".SP_PID,
                                DB := "Control_NAD".DB_PID,
                                KP := "Control_NAD".KP_PID,
                                TI := "Control_NAD".TI_PID,
                                TD := "Control_NAD".TD_PID,
                                CYCLE := 100,
                                FMT := "Control_NAD".FMT_PID,
                                DT_MIN := "Control_NAD".DT_MIN_PID,
                                AUTO := ("Control_NAD".Mode AND "Control_NAD".Mode_from_PLC AND NOT "dP_furnace_boiler".Error_sensor),
                                MORE := ((NOT "Control_NAD".Mode AND "Control_NAD".Manual_open) OR ("Control_NAD".Mode AND "Control_NAD".Manual_open_from_PLC)),
                                LESS := ((NOT "Control_NAD".Mode AND "Control_NAD".Manual_close) OR ("Control_NAD".Mode AND "Control_NAD".Manual_close_from_PLC)),
                                Hold := false,
                                GAP := "Control_NAD".GAP,
                                PLUS := "NAD_control_open".Value,
                                MINUS := "NAD_control_close".Value);
       ELSE    //ручной режим
           "PID_impulse_NAD_DB"(DIR := FALSE,
                                PV := "dP_furnace_boiler".Value,
                                SP := "dP_furnace_boiler".Value,
                                DB := "Control_NAD".DB_PID,
                                KP := "Control_NAD".KP_PID,
                                TI := "Control_NAD".TI_PID,
                                TD := "Control_NAD".TD_PID,
                                CYCLE := 100,
                                FMT := "Control_NAD".FMT_PID,
                                DT_MIN := "Control_NAD".DT_MIN_PID,
                                AUTO := ("Control_NAD".Mode AND "Control_NAD".Mode_from_PLC AND NOT "dP_furnace_boiler".Error_sensor),
                                MORE := ((NOT "Control_NAD".Mode AND "Control_NAD".Manual_open) OR ("Control_NAD".Mode AND "Control_NAD".Manual_open_from_PLC)),
                                LESS := ((NOT "Control_NAD".Mode AND "Control_NAD".Manual_close) OR ("Control_NAD".Mode AND "Control_NAD".Manual_close_from_PLC)),
                                Hold := false,
                                GAP := "Control_NAD".GAP,
                                PLUS := "NAD_control_open".Value,
                                MINUS := "NAD_control_close".Value);
       END_IF;
   ELSE
       //при переводе БРУ в ручной режим
       "NAD_control_open".Value := FALSE;
       "NAD_control_close".Value := FALSE;
       "Control_NAD".Manual_open := FALSE;
       "Control_NAD".Manual_close := FALSE;
       "PID_impulse_NAD_DB"(DIR := FALSE,
                            PV := "dP_furnace_boiler".Value,
                            SP := "dP_furnace_boiler".Value,
                            DB := "Control_NAD".DB_PID,
                            KP := "Control_NAD".KP_PID,
                            TI := "Control_NAD".TI_PID,
                            TD := "Control_NAD".TD_PID,
                            CYCLE := 100,
                            FMT := "Control_NAD".FMT_PID,
                            DT_MIN := "Control_NAD".DT_MIN_PID,
                            AUTO := FALSE,
                            MORE := FALSE,
                            LESS := FALSE,
                            Hold := false,
                            GAP := "Control_NAD".GAP,
                            PLUS := "NAD_control_open".Value,
                            MINUS := "NAD_control_close".Value);
   END_IF;

   (*ЗДГ*)
   //Проверка и сброс ручных команд
   //Сброс всех команд при автоматическом режиме
   IF "Control_ZDG".Mode THEN
       "Control_ZDG".Manual_open := FALSE;
       "Control_ZDG".Manual_close := FALSE;
       "Control_ZDG".Manual_stop := FALSE;
   END_IF;
   //сброс обеих команд при их одновременном наличии
   IF "Control_ZDG".Manual_open AND "Control_ZDG".Manual_close THEN
       "Control_ZDG".Manual_open := FALSE;
       "Control_ZDG".Manual_close := FALSE;
       "Control_ZDG".Manual_stop := TRUE;
   END_IF;
   //сброс ручных команд при начале движения
   IF "ZDG_opening".Value OR "ZDG_closing".Value THEN
       "Control_ZDG".Manual_open := FALSE;
       "Control_ZDG".Manual_close := FALSE;
   END_IF;
   //сброс команды стоп при окончаниии движения
   IF NOT "ZDG_opening".Value AND NOT "ZDG_closing".Value THEN
       "Control_ZDG".Manual_stop := FALSE;
   END_IF;
   //сброс команды открыть при полном открытии или запрете
   IF NOT "ZDG_no_open".Value OR "ZDG_control_disable_open".Value THEN
       "Control_ZDG".Manual_open := FALSE;
   END_IF;
   //сброс команды закрыть при полном закрытии
   IF NOT "ZDG_no_close".Value THEN
       "Control_ZDG".Manual_close := FALSE;
   END_IF;
   //Проверка и сброс автоматических команд
   //сброс обеих команд при их одновременном наличии
   IF "Control_ZDG".Avto_open AND "Control_ZDG".Avto_close THEN
       "Control_ZDG".Avto_open := FALSE;
       "Control_ZDG".Avto_close := FALSE;
       "Control_ZDG".Avto_stop := TRUE;
   END_IF;
   //сброс команд при начале движения
   IF "ZDG_opening".Value OR "ZDG_closing".Value THEN
       "Control_ZDG".Avto_open := FALSE;
       "Control_ZDG".Avto_close := FALSE;
   END_IF;
   //сброс команды стоп при окончаниии движения
   IF NOT "ZDG_opening".Value AND NOT "ZDG_closing".Value THEN
       "Control_ZDG".Avto_stop := FALSE;
   END_IF;
   //сброс команды открыть при полном открытии или запрете
   IF NOT "ZDG_no_open".Value OR "ZDG_control_disable_open".Value THEN
       "Control_ZDG".Avto_open := FALSE;
   END_IF;
   //сброс команды закрыть при полном закрытии
   IF NOT "ZDG_no_close".Value THEN
       "Control_ZDG".Avto_close := FALSE;
   END_IF;
   //управление
   IF "Control_ZDG".Mode THEN
       // автоматический режим
       "ZDG_control_open".Value := "Control_ZDG".Avto_open;
       "ZDG_control_close".Value := "Control_ZDG".Avto_close;
       "ZDG_control_stop".Value := "Control_ZDG".Avto_stop;
   ELSE
       //ручной режим
       "ZDG_control_open".Value := "Control_ZDG".Manual_open;
       "ZDG_control_close".Value := "Control_ZDG".Manual_close;
       "ZDG_control_stop".Value := "Control_ZDG".Manual_stop;
   END_IF;
   //Управление запретом открытия
   IF "Technology".Regim <> 1 AND
       ("PZK1_open".Value OR                                  //ПЗК1 открыт
       ("PZK2_open".Value OR "PZK2_not_close".Value) OR     //ПЗК2 открыт
       //("Sensors".Q_water_boiler_min.Value AND NOT "Protections".BLOCK_Q_water_boiler_min) OR    //нет расхода воды
       "L_water_min".Value OR  //минимальный уровень воды в барабане
       (NOT "DV_invertor_on".Value AND NOT "DV_powergrid_on".Value)) THEN //ДВ  
       "ZDG_control_disable_open".Value := TRUE;
   ELSE
       "ZDG_control_disable_open".Value := FALSE;
   END_IF;

   (*КБ*)
   //при переходе из автоматического в ручной режим управления в ручную команду копируем текущее положение
   "F_TRIG_KB_DB"(CLK := "Control_KB".Mode,
                  Q => "FRONT".KB_mode);
   IF "FRONT".KB_mode THEN
       "Control_KB".Manual_close := "KB_close".Value;
   END_IF;
   //управление
   IF "Control_KB".Mode THEN
       // автоматический режим
       "KB_control_close".Value := "Control_KB".Avto_close;
   ELSE
       //ручной режим
       "KB_control_close".Value := "Control_KB".Manual_close;
   END_IF;

   (*КО*)
   //при переходе из автоматического в ручной режим управления в ручную команду копируем текущее положение
   "F_TRIG_KO_DB"(CLK := "Control_KO".Mode,
                  Q => "FRONT".KO_mode);
   IF "FRONT".KO_mode THEN
       "Control_KO".Manual_open := "KO_open".Value;
   END_IF;
   //управление
   IF "Control_KO".Mode THEN
       // автоматический режим
       "KO_control_open".Value := "Control_KO".Avto_open;
   ELSE
       //ручной режим
       "KO_control_open".Value := "Control_KO".Manual_open;
   END_IF;

   (*КЗ*)
   //при переходе из автоматического в ручной режим управления в ручную команду копируем текущее положение
   "F_TRIG_KZ_DB"(CLK := "Control_KZ".Mode,
                  Q => "FRONT".KZ_mode);
   IF "FRONT".KZ_mode THEN
       "Control_KZ".Manual_open := "KZ_open".Value;
   END_IF;
   //закрытие клапана запальника по таймеру
   "TON_close_KZ_DB".TON(IN := "Timer".close_KZ_IN,
                         PT := T#25s,
                         Q => "Timer".close_KZ_Q);
   IF "Timer".close_KZ_Q THEN
       "Timer".close_KZ_IN := FALSE;
       "Control_KZ".Avto_open := FALSE;
   END_IF;
   //управление
   IF "Control_KZ".Mode THEN
       // автоматический режим
       "KZ_control_open".Value := "Control_KZ".Avto_open;
   ELSE
       //ручной режим
       "KZ_control_open".Value := "Control_KZ".Manual_open;
   END_IF;

   (*ИВН*)
   //при переходе из автоматического в ручной режим управления в ручную команду копируем текущую команду
   "F_TRIG_IVN_DB"(CLK := "Control_IVN".Mode,
                   Q => "FRONT".IVN_mode);
   IF "FRONT".IVN_mode THEN
       "Control_IVN".Manual_on := "Control_IVN".Avto_on;
   END_IF;
   //сброс автоматической команды на включения через 6 секунд
   "TON_avto_reset_IVN_DB".TON(IN := "IVN_control_on".Value,
                               PT := T#6s,
                               Q => "Timer".avto_reset_IVN_Q);
   IF "Timer".avto_reset_IVN_Q THEN
       "Control_IVN".Avto_on := FALSE;
   END_IF;
   //управление
   IF "Control_IVN".Mode THEN
       // автоматический режим
       "IVN_control_on".Value := "Control_IVN".Avto_on;
   ELSE
       //ручной режим
       "IVN_control_on".Value := "Control_IVN".Manual_on;
   END_IF;

   (*ПЗК1*)
   //при переходе из автоматического в ручной режим управления в ручную команду копируем текущее положение
   "F_TRIG_PZK1_DB"(CLK := "Control_PZK1".Mode,
                    Q => "FRONT".PZK1_mode);
   IF "FRONT".PZK1_mode THEN
       "Control_PZK1".Manual_open := "PZK1_open".Value;
   END_IF;
   IF "Control_PZK1".Mode THEN
       // автоматический режим
       "PZK1_control_open".Value := "Control_PZK1".Avto_open;
   ELSE
       //ручной режим
       "PZK1_control_open".Value := "Control_PZK1".Manual_open;
   END_IF;

   (*ПЗК2*)
   //при переходе из автоматического в ручной режим управления в ручную команду копируем текущее положение
   "F_TRIG_PZK2_DB"(CLK := "Control_PZK2".Mode,
                    Q => "FRONT".PZK2_mode);
   IF "FRONT".PZK2_mode THEN
       "Control_PZK2".Manual_open := "PZK2_open".Value;
   END_IF;
   IF "Control_PZK2".Mode THEN
       // автоматический режим
       "PZK2_control_open".Value := "Control_PZK2".Avto_open;
   ELSE
       //ручной режим
       "PZK2_control_open".Value := "Control_PZK2".Manual_open;
   END_IF;

   (*ЗДСВ перед котлом*)
   //Проверка и сброс ручных команд
   //Сброс всех команд при автоматическом режиме
   IF "Control_ZDSV_before_boiler".Mode THEN
       "Control_ZDSV_before_boiler".Manual_open := FALSE;
       "Control_ZDSV_before_boiler".Manual_close := FALSE;
       "Control_ZDSV_before_boiler".Manual_stop := FALSE;
   END_IF;
   //сброс обеих команд при их одновременном наличии
   IF "Control_ZDSV_before_boiler".Manual_open AND "Control_ZDSV_before_boiler".Manual_close THEN
       "Control_ZDSV_before_boiler".Manual_open := FALSE;
       "Control_ZDSV_before_boiler".Manual_close := FALSE;
       "Control_ZDSV_before_boiler".Manual_stop := TRUE;
   END_IF;
   //сброс ручных команд при начале движения
   IF "ZDSV_before_boiler_opening".Value OR "ZDSV_before_boiler_closing".Value THEN
       "Control_ZDSV_before_boiler".Manual_open := FALSE;
       "Control_ZDSV_before_boiler".Manual_close := FALSE;
   END_IF;
   //сброс команды стоп при окончаниии движения
   IF NOT "ZDSV_before_boiler_opening".Value AND NOT "ZDSV_before_boiler_closing".Value THEN
       "Control_ZDSV_before_boiler".Manual_stop := FALSE;
   END_IF;
   //сброс команды открыть при полном открытии
   IF NOT "ZDSV_before_boiler_no_open".Value THEN
       "Control_ZDSV_before_boiler".Manual_open := FALSE;
   END_IF;
   //сброс команды закрыть при полном закрытии или запрете
   IF NOT "ZDSV_before_boiler_no_close".Value OR "ZDSV_before_boiler_control_disable_close".Value THEN
       "Control_ZDSV_before_boiler".Manual_close := FALSE;
   END_IF;
   //Проверка и сброс автоматических команд
   //сброс обеих команд при их одновременном наличии
   IF "Control_ZDSV_before_boiler".Avto_open AND "Control_ZDSV_before_boiler".Avto_close THEN
       "Control_ZDSV_before_boiler".Avto_open := FALSE;
       "Control_ZDSV_before_boiler".Avto_close := FALSE;
       "Control_ZDSV_before_boiler".Avto_stop := TRUE;
   END_IF;
   //сброс ручных команд при начале движения
   IF "ZDSV_before_boiler_opening".Value OR "ZDSV_before_boiler_closing".Value THEN
       "Control_ZDSV_before_boiler".Avto_open := FALSE;
       "Control_ZDSV_before_boiler".Avto_close := FALSE;
   END_IF;
   //сброс команды стоп при окончаниии движения
   IF NOT "ZDSV_before_boiler_opening".Value AND NOT "ZDSV_before_boiler_closing".Value THEN
       "Control_ZDSV_before_boiler".Avto_stop := FALSE;
   END_IF;
   //сброс команды открыть при полном открытии
   IF NOT "ZDSV_before_boiler_no_open".Value THEN
       "Control_ZDSV_before_boiler".Avto_open := FALSE;
   END_IF;
   //сброс команды закрыть при полном закрытии или запрете
   IF NOT "ZDSV_before_boiler_no_close".Value OR "ZDSV_before_boiler_control_disable_close".Value THEN
       "Control_ZDSV_before_boiler".Avto_close := FALSE;
   END_IF;
   //управление
   IF "Control_ZDSV_before_boiler".Mode THEN
       // автоматический режим
       "ZDSV_before_boiler_control_open".Value := "Control_ZDSV_before_boiler".Avto_open;
       "ZDSV_before_boiler_control_close".Value := "Control_ZDSV_before_boiler".Avto_close;
       "ZDSV_before_boiler_control_stop".Value := "Control_ZDSV_before_boiler".Avto_stop;
   ELSE
       //ручной режим
       "ZDSV_before_boiler_control_open".Value := "Control_ZDSV_before_boiler".Manual_open;
       "ZDSV_before_boiler_control_close".Value := "Control_ZDSV_before_boiler".Manual_close;
       "ZDSV_before_boiler_control_stop".Value := "Control_ZDSV_before_boiler".Manual_stop;
   END_IF;
   //Управление запретом закрытия
   IF "ZDG_no_close".Value OR                              //ЗДГ не закрыта
       ("L_water_min".Value AND NOT "Protections_BLOCK".L_water_min) THEN               //Мало воды в барабане
       "ZDSV_before_boiler_control_disable_close".Value := TRUE;
   ELSE
       "ZDSV_before_boiler_control_disable_close".Value := FALSE;
   END_IF;

   (*ГПЗ*)
   //Проверка и сброс ручных команд
   //Сброс всех команд при автоматическом режиме
   IF "Control_GPZ".Mode THEN
       "Control_GPZ".Manual_open := FALSE;
       "Control_GPZ".Manual_close := FALSE;
       "Control_GPZ".Manual_stop := FALSE;
   END_IF;
   //сброс обоих команд при их одновременном наличии
   IF "Control_GPZ".Manual_open AND "Control_GPZ".Manual_close THEN
       "Control_GPZ".Manual_open := FALSE;
       "Control_GPZ".Manual_close := FALSE;
       "Control_GPZ".Manual_stop := TRUE;
   END_IF;
   //сброс ручных команд при начале движения
   IF "GPZ_opening".Value OR "GPZ_closing".Value THEN
       "Control_GPZ".Manual_open := FALSE;
       "Control_GPZ".Manual_close := FALSE;
   END_IF;
   //сброс команды стоп при окончаниии движения
   IF NOT "GPZ_opening".Value AND NOT "GPZ_closing".Value THEN
       "Control_GPZ".Manual_stop := FALSE;
   END_IF;
   //сброс команды открыть при полном открытии
   IF NOT "GPZ_no_open".Value THEN
       "Control_GPZ".Manual_open := FALSE;
   END_IF;
   //сброс команды закрыть при полном закрытии или запрете
   IF NOT "GPZ_no_close".Value OR "GPZ_control_disable_close".Value THEN
       "Control_GPZ".Manual_close := FALSE;
   END_IF;
   //Проверка и сброс автоматических команд
   //сброс обоих команд при их одновременном наличии
   IF "Control_GPZ".Avto_open AND "Control_GPZ".Avto_close THEN
       "Control_GPZ".Avto_open := FALSE;
       "Control_GPZ".Avto_close := FALSE;
       "Control_GPZ".Avto_stop := TRUE;
   END_IF;
   //сброс ручных команд при начале движения
   IF "GPZ_opening".Value OR "GPZ_closing".Value THEN
       "Control_GPZ".Avto_open := FALSE;
       "Control_GPZ".Avto_close := FALSE;
   END_IF;
   //сброс команды стоп при окончаниии движения
   IF NOT "GPZ_opening".Value AND NOT "GPZ_closing".Value THEN
       "Control_GPZ".Avto_stop := FALSE;
   END_IF;
   //сброс команды открыть при полном открытии
   IF NOT "GPZ_no_open".Value THEN
       "Control_GPZ".Avto_open := FALSE;
   END_IF;
   //сброс команды закрыть при полном закрытии или запрете
   IF NOT "GPZ_no_close".Value OR "GPZ_control_disable_close".Value THEN
       "Control_GPZ".Avto_close := FALSE;
   END_IF;
   //управление
   IF "Control_GPZ".Mode THEN
       // автоматический режим
       "GPZ_control_open".Value := "Control_GPZ".Avto_open;
       "GPZ_control_close".Value := "Control_GPZ".Avto_close;
       "GPZ_control_stop".Value := "Control_GPZ".Avto_stop;
   ELSE
       //ручной режим
       "GPZ_control_open".Value := "Control_GPZ".Manual_open;
       "GPZ_control_close".Value := "Control_GPZ".Manual_close;
       "GPZ_control_stop".Value := "Control_GPZ".Manual_stop;
   END_IF;
   //Управление запретом закрытия
   IF //"GPZ_no_close".Value OR       //ГПЗ не закрыта
       "Technology".Regim <> 1 AND
       (("P_steam_max".Value AND NOT "Protections_BLOCK".P_steam_max)) THEN     //P в барабане котла max 
       "GPZ_control_disable_close".Value := TRUE;
   ELSE
       "GPZ_control_disable_close".Value := FALSE;
   END_IF;
   //Автоматическое управление
   "Timer_сlose_GPZ_DB".TON(IN := "Timer".Close_GPZ_IN,
                            PT := "Timer".Close_GPZ_PT,
                            Q => "Timer".Close_GPZ_Q);

   IF NOT "PZK2_not_close".Value AND NOT "PZK2_open".Value THEN
       "Timer".Close_GPZ_IN := TRUE;
   ELSE
       "Timer".Close_GPZ_IN := FALSE;
   END_IF;
   IF "Timer".Close_GPZ_Q AND "GPZ_no_close".Value THEN
       "Control_GPZ".Avto_close := TRUE;
   ELSE
       "Control_GPZ".Avto_close := FALSE;
   END_IF;

   (*ДВ*)
   //Проверка и сброс ручных команд
   //Сброс команд при автоматическом режиме
   IF "Control_DV".Mode THEN
       "Control_DV".Manual_Start := FALSE;
       "Control_DV".Manual_Stop := FALSE;
   END_IF;
   "F_TRIG_DV_DB"(CLK := "Control_DV".Mode,
                  Q => "FRONT".DV_mode);
   IF "FRONT".DV_mode THEN
       "Control_DV".Manual_frequency := "PID_analog_DV_DB".OUT;
   END_IF;
   //обеих команд при их одновременном наличии или отсутствии дистанционного режима
   IF ("Control_DV".Manual_Start AND "Control_DV".Manual_Stop) OR
       NOT "DV_dist_control".Value THEN
       "Control_DV".Manual_Start := FALSE;
       "Control_DV".Manual_Stop := FALSE;
   END_IF;
   //Подача команды на отключение при аварии ПЧ
   IF NOT "Control_DV".Mode AND "Warning".DV_invertor_alarm AND "DV_invertor_on".Value THEN
       "Control_DV".Manual_Stop := TRUE;
   END_IF;
   //сброс команды пуск после включения
   IF "DV_invertor_on".Value OR "DV_powergrid_on".Value THEN
       "Control_DV".Manual_Start := FALSE;
   END_IF;
   //сброс команды пуск и подача команды стоп при отключенном ДС
   (*IF NOT "Sensors".DS_invertor_on.Value AND NOT "Sensors".DS_powergrid_on.Value THEN
       "Control_DV".Manual_Start := FALSE;
   END_IF;*)
   //сброс команды стоп после отключения
   IF NOT "DV_invertor_on".Value AND NOT "DV_powergrid_on".Value THEN
       "Control_DV".Manual_Stop := FALSE;
   END_IF;
   //Проверка и сброс автоматических команд
   //сброс обеих команд при их одновременном наличии
   IF "Control_DV".Avto_Start AND "Control_DV".Avto_Stop THEN
       "Control_DV".Avto_Start := FALSE;
       "Control_DV".Avto_Stop := FALSE;
   END_IF;
   //Подача команды на отключение при аварии ПЧ
   IF "Control_DV".Mode AND "Warning".DV_invertor_alarm AND "DV_invertor_on".Value THEN
       "Control_DV".Avto_Stop := TRUE;
   END_IF;
   IF "Warning".DV_invertor_alarm AND "DV_invertor_mode".Value THEN
       "Control_DV".Avto_Start := FALSE;
   END_IF;
   //сброс команды пуск после включения
   IF "DV_invertor_on".Value OR "DV_powergrid_on".Value THEN
       "Control_DV".Avto_Start := FALSE;
   END_IF;
   //сброс команды стоп после отключения
   IF NOT "DV_invertor_on".Value AND NOT "DV_powergrid_on".Value THEN
       "Control_DV".Avto_Stop := FALSE;
   END_IF;
   //управление
   IF "DV_dist_control".Value THEN    //Управление «Дистанционный» ДВ
       //включение
       IF "Control_DV".Mode THEN
           // автоматический режим
           "DV_control_start".Value := "Control_DV".Avto_Start;
           "DV_control_stop".Value := "Control_DV".Avto_Stop;
       ELSE
           //ручной режим
           "DV_control_start".Value := "Control_DV".Manual_Start;
           "DV_control_stop".Value := "Control_DV".Manual_Stop;
       END_IF;
       //частота
       IF "DV_invertor_mode".Value THEN    //Режим "ПЧ" ДВ
           "PID_analog_DV_DB"(AUTO := ("Control_DV".Mode AND "Control_DV".Mode_from_PLC AND NOT "P_air_burner".Error_sensor),
                              DIR := TRUE,
                              PV := "P_air_burner".Value,
                              SP := "Control_DV".SP_PID,
                              DB := "Control_DV".DB_PID,
                              KP := "Control_DV".KP_PID,
                              TI := "Control_DV".TI_PID,
                              TD := "Control_DV".TD_PID,
                              CYCLE := 100,
                              Hold := false,
                              OUT_MIN := 7.0,
                              OUT_MAX := "DV_control_frequency".HL_control_signal_new,
                              OUT := "DV_control_frequency".Value);
           IF "Control_DV".Mode THEN
               "PID_analog_DV_DB".OUT_MAN := "Control_DV".Manual_frequency_from_PLC;
           ELSE
               "PID_analog_DV_DB".OUT_MAN := "Control_DV".Manual_frequency;
           END_IF;
       ELSE
           //"PID_analog_DV_DB".Hold := TRUE;
           "DV_control_frequency".Value := 0.0;
       END_IF;
   ELSE
       "DV_control_start".Value := FALSE;
       "DV_control_stop".Value := FALSE;
       "DV_control_frequency".Value := 0.0;
   END_IF;

   (*ДС*)
   //Проверка и сброс ручных команд
   //Сброс команд при автоматическом режиме
   IF "Control_DS".Mode THEN
       "Control_DS".Manual_Start := FALSE;
       "Control_DS".Manual_Stop := FALSE;
   END_IF;
   "F_TRIG_DS_DB"(CLK := "Control_DS".Mode,
                  Q => "FRONT".DS_mode);
   IF "FRONT".DS_mode THEN
       "Control_DS".Manual_frequency := "PID_analog_DS_DB".OUT;
   END_IF;
   //сброс обоих команд при их одновременном наличии или отсутствии дистанционного режима
   IF ("Control_DS".Manual_Start AND "Control_DS".Manual_Stop) OR
       NOT "DS_dist_control".Value THEN
       "Control_DS".Manual_Start := FALSE;
       "Control_DS".Manual_Stop := FALSE;
   END_IF;
   //Подача команды на отключение при аварии ПЧ
   IF NOT "Control_DS".Mode AND "Warning".DS_invertor_alarm AND "DS_invertor_on".Value THEN
       "Control_DS".Manual_Stop := TRUE;
   END_IF;
   //сброс команды пуск после включения
   IF "DS_invertor_on".Value OR "DS_powergrid_on".Value THEN
       "Control_DS".Manual_Start := FALSE;
   END_IF;
   //сброс команды стоп после отключения
   IF NOT "DS_invertor_on".Value AND NOT "DS_powergrid_on".Value THEN
       "Control_DS".Manual_Stop := FALSE;
   END_IF;
   //Проверка и сброс автоматических команд
   //сброс обоих команд при их одновременном наличии
   IF "Control_DS".Avto_Start AND "Control_DS".Avto_Stop THEN
       "Control_DS".Avto_Start := FALSE;
       "Control_DS".Avto_Stop := FALSE;
   END_IF;
   //Подача команды на отключение при аварии ПЧ
   IF "Control_DS".Mode AND "Warning".DS_invertor_alarm AND "DS_invertor_on".Value THEN
       "Control_DS".Avto_Stop := TRUE;
   END_IF;
   IF "Warning".DS_invertor_alarm AND "DS_invertor_mode".Value THEN
       "Control_DS".Avto_Start := FALSE;
   END_IF;
   //сброс команды пуск после включения
   IF "DS_invertor_on".Value OR "DS_powergrid_on".Value THEN
       "Control_DS".Avto_Start := FALSE;
   END_IF;
   //сброс команды стоп после отключения
   IF NOT "DS_invertor_on".Value AND NOT "DS_powergrid_on".Value THEN
       "Control_DS".Avto_Stop := FALSE;
   END_IF;
   //управление
   IF "DS_dist_control".Value THEN    //Управление «Дистанционный» ДС
       //включение
       IF "Control_DS".Mode THEN
           // автоматический режим
           "DS_control_start".Value := "Control_DS".Avto_Start;
           "DS_control_stop".Value := "Control_DS".Avto_Stop;
       ELSE
           //ручной режим
           "DS_control_start".Value := "Control_DS".Manual_Start;
           "DS_control_stop".Value := "Control_DS".Manual_Stop;
       END_IF;
       //частота
       IF "DS_invertor_mode".Value THEN    //Режим "ПЧ" ДС
           "PID_analog_DS_DB"(AUTO := ("Control_DS".Mode AND "Control_DS".Mode_from_PLC AND NOT "dP_furnace_boiler".Error_sensor),
                              DIR := FALSE,
                              PV := "dP_furnace_boiler".Value,
                              SP := "Control_DS".SP_PID,
                              DB := "Control_DS".DB_PID,
                              KP := "Control_DS".KP_PID,
                              TI := "Control_DS".TI_PID,
                              TD := "Control_DS".TD_PID,
                              CYCLE := 100,
                              Hold := false,
                              OUT_MIN := 7.0,
                              OUT_MAX := "DS_control_frequency".HL_control_signal_new,
                              OUT := "DS_control_frequency".Value);
           IF "Control_DS".Mode THEN
               "PID_analog_DS_DB".OUT_MAN := "Control_DS".Manual_frequency_from_PLC;
           ELSE
               "PID_analog_DS_DB".OUT_MAN := "Control_DS".Manual_frequency;
           END_IF;
       ELSE
           //"PID_analog_DS_DB".Hold := TRUE;
           "DS_control_frequency".Value := 0.0;
       END_IF;
   ELSE
       "DS_control_start".Value := FALSE;
       "DS_control_stop".Value := FALSE;
       "DS_control_frequency".Value := 0.0;
   END_IF;
END_FUNCTION

ORGANIZATION_BLOCK "Main"   // OB1, LAD, ProgramCycle
TITLE = "Main Program Sweep (Cycle)"
{ S7_Optimized_Access := 'TRUE' }
VERSION : 0.1
   VAR_INPUT
      Initial_Call : Bool;   // Initial call of this OB
      Remanence : Bool;   // =True, if remanent data are available
   END_VAR
BEGIN

REGION Network 1
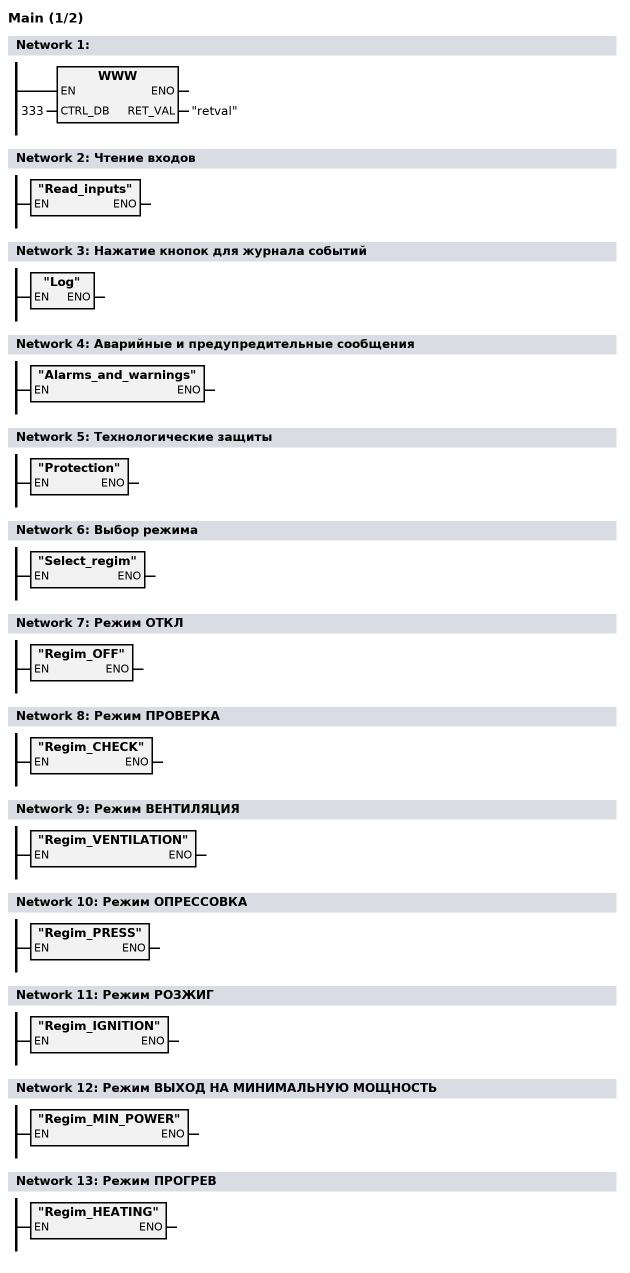
   "retval" := WWW(CTRL_DB := 333);
END_REGION

REGION Network 2: Чтение входов
   RUNG wire#powerrail
      "Read_inputs"()
   END_RUNG
   // the same network as SCL:
   "Read_inputs"();
END_REGION

REGION Network 3: Нажатие кнопок для журнала событий
   RUNG wire#powerrail
      "Log"()
   END_RUNG
   // the same network as SCL:
   "Log"();
END_REGION

REGION Network 4: Аварийные и предупредительные сообщения
   RUNG wire#powerrail
      "Alarms_and_warnings"()
   END_RUNG
   // the same network as SCL:
   "Alarms_and_warnings"();
END_REGION

REGION Network 5: Технологические защиты
   RUNG wire#powerrail
      "Protection"()
   END_RUNG
   // the same network as SCL:
   "Protection"();
END_REGION

REGION Network 6: Выбор режима
   RUNG wire#powerrail
      "Select_regim"()
   END_RUNG
   // the same network as SCL:
   "Select_regim"();
END_REGION

REGION Network 7: Режим ОТКЛ
   RUNG wire#powerrail
      "Regim_OFF"()
   END_RUNG
   // the same network as SCL:
   "Regim_OFF"();
END_REGION

REGION Network 8: Режим ПРОВЕРКА
   RUNG wire#powerrail
      "Regim_CHECK"()
   END_RUNG
   // the same network as SCL:
   "Regim_CHECK"();
END_REGION

REGION Network 9: Режим ВЕНТИЛЯЦИЯ
   RUNG wire#powerrail
      "Regim_VENTILATION"()
   END_RUNG
   // the same network as SCL:
   "Regim_VENTILATION"();
END_REGION

REGION Network 10: Режим ОПРЕССОВКА
   RUNG wire#powerrail
      "Regim_PRESS"()
   END_RUNG
   // the same network as SCL:
   "Regim_PRESS"();
END_REGION

REGION Network 11: Режим РОЗЖИГ
   RUNG wire#powerrail
      "Regim_IGNITION"()
   END_RUNG
   // the same network as SCL:
   "Regim_IGNITION"();
END_REGION

REGION Network 12: Режим ВЫХОД НА МИНИМАЛЬНУЮ МОЩНОСТЬ
   RUNG wire#powerrail
      "Regim_MIN_POWER"()
   END_RUNG
   // the same network as SCL:
   "Regim_MIN_POWER"();
END_REGION

REGION Network 13: Режим ПРОГРЕВ
   RUNG wire#powerrail
      "Regim_HEATING"()
   END_RUNG
   // the same network as SCL:
   "Regim_HEATING"();
END_REGION

REGION Network 14: Режим РАБОТА
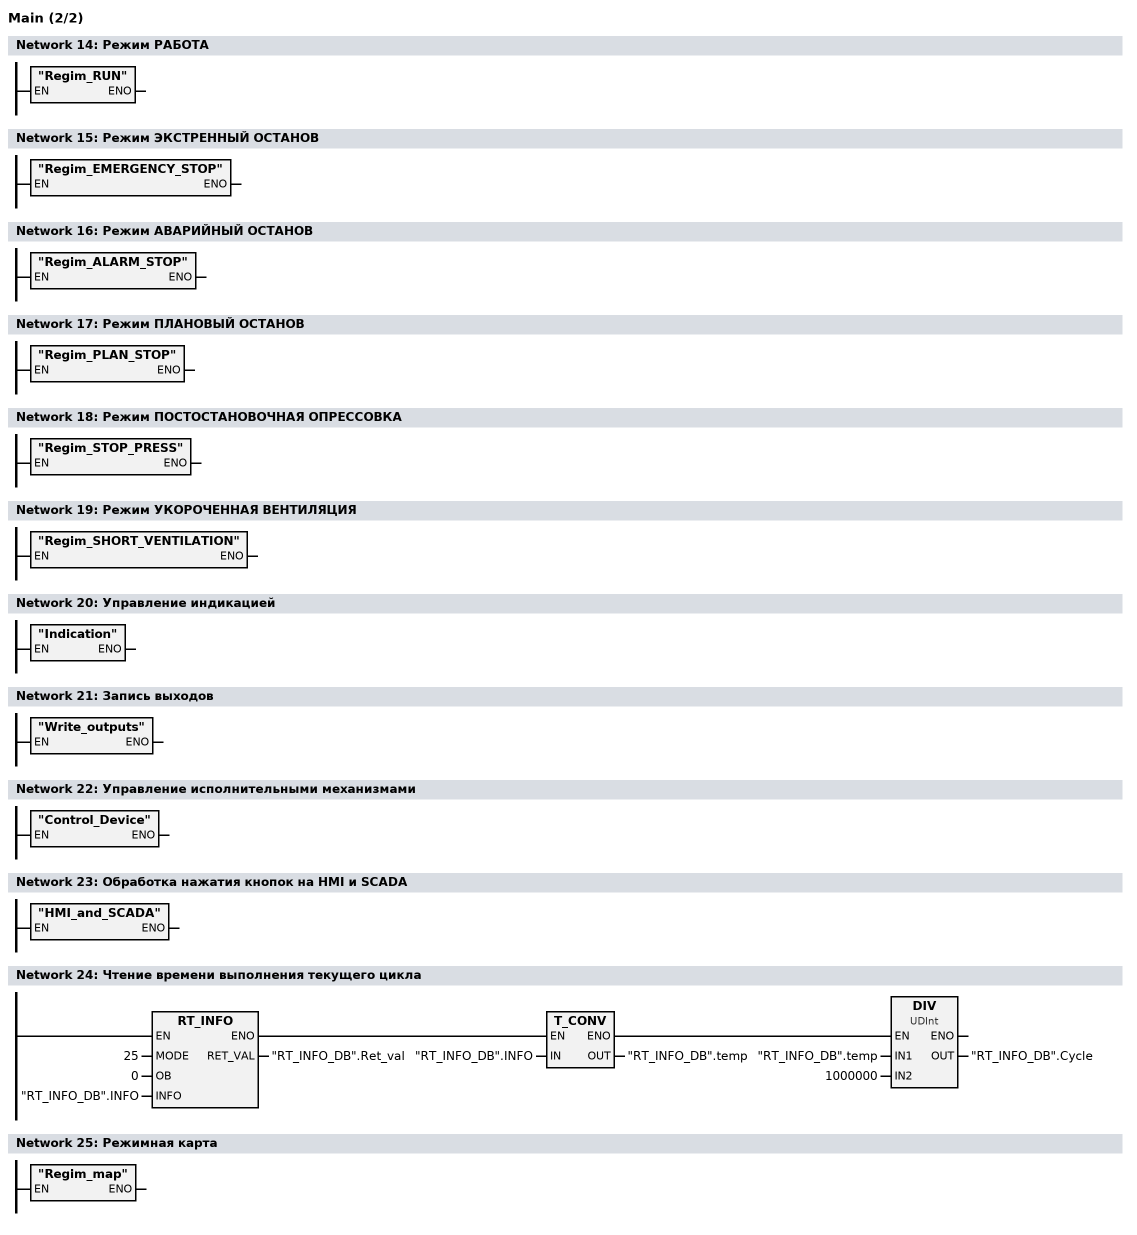
   RUNG wire#powerrail
      "Regim_RUN"()
   END_RUNG
   // the same network as SCL:
   "Regim_RUN"();
END_REGION

REGION Network 15: Режим ЭКСТРЕННЫЙ ОСТАНОВ
   RUNG wire#powerrail
      "Regim_EMERGENCY_STOP"()
   END_RUNG
   // the same network as SCL:
   "Regim_EMERGENCY_STOP"();
END_REGION

REGION Network 16: Режим АВАРИЙНЫЙ ОСТАНОВ
   RUNG wire#powerrail
      "Regim_ALARM_STOP"()
   END_RUNG
   // the same network as SCL:
   "Regim_ALARM_STOP"();
END_REGION

REGION Network 17: Режим ПЛАНОВЫЙ ОСТАНОВ
   RUNG wire#powerrail
      "Regim_PLAN_STOP"()
   END_RUNG
   // the same network as SCL:
   "Regim_PLAN_STOP"();
END_REGION

REGION Network 18: Режим ПОСТОСТАНОВОЧНАЯ ОПРЕССОВКА
   RUNG wire#powerrail
      "Regim_STOP_PRESS"()
   END_RUNG
   // the same network as SCL:
   "Regim_STOP_PRESS"();
END_REGION

REGION Network 19: Режим УКОРОЧЕННАЯ ВЕНТИЛЯЦИЯ
   RUNG wire#powerrail
      "Regim_SHORT_VENTILATION"()
   END_RUNG
   // the same network as SCL:
   "Regim_SHORT_VENTILATION"();
END_REGION

REGION Network 20: Управление индикацией
   RUNG wire#powerrail
      "Indication"()
   END_RUNG
   // the same network as SCL:
   "Indication"();
END_REGION

REGION Network 21: Запись выходов
   RUNG wire#powerrail
      "Write_outputs"()
   END_RUNG
   // the same network as SCL:
   "Write_outputs"();
END_REGION

REGION Network 22: Управление исполнительными механизмами
   RUNG wire#powerrail
      "Control_Device"()
   END_RUNG
   // the same network as SCL:
   "Control_Device"();
END_REGION

REGION Network 23: Обработка нажатия кнопок на HMI и SCADA
   RUNG wire#powerrail
      "HMI_and_SCADA"()
   END_RUNG
   // the same network as SCL:
   "HMI_and_SCADA"();
END_REGION

REGION Network 24: Чтение времени выполнения текущего цикла
   // ENO of a box is taken as its EN; it also drops when the box reports an error
   "RT_INFO_DB".Ret_val := RT_INFO(MODE := 25, OB := 0, INFO := "RT_INFO_DB".INFO);
   "RT_INFO_DB".temp := T_CONV(IN := "RT_INFO_DB".INFO);
   "RT_INFO_DB".Cycle := "RT_INFO_DB".temp / 1000000;
END_REGION

REGION Network 25: Режимная карта
   RUNG wire#powerrail
      "Regim_map"()
   END_RUNG
   // the same network as SCL:
   "Regim_map"();
END_REGION
END_ORGANIZATION_BLOCK

// folder: Regims

FUNCTION "Regim_VENTILATION" : Void   // FC13, SCL
{ S7_Optimized_Access := 'TRUE' }
VERSION : 0.1
BEGIN
   (*Режим ВЕНТИЛЯЦИЯ*)
   (*таймеры*)
   "Timer_VENTILATION_temp_DB".TON(IN := "Timer".VENTILATION_temp_IN,
                                   PT := "Timer".VENTILATION_temp_PT,
                                   Q => "Timer".VENTILATION_temp_Q);
   "Timer_VENTILATION_DB".TONR(IN := "Timer".VENTILATION_IN,
                               R := "Timer".VENTILATION_R,
                               PT := "Timer".VENTILATION_PT,
                               Q => "Timer".VENTILATION_Q);
   (*процесс*)
   IF "Technology".Regim = 3 THEN
       CASE "Technology".Regim_ventilation_step OF
           0:  //проверяем положение ИМ по газу
               "Technology".Regim_ventilation_step := 1;

           1:  //снимаем защиту Повышение давления газа перед БГ
               "Alarm_Enable".P_gas_before_BG_max := FALSE;
               //снимаем защиту Понижение давления газа перед БГ
               "Alarm_Enable".P_gas_before_BG_min := FALSE;
               //перевод клапанов по газу в исходное состояние
               "Control_PZK1".Mode := TRUE;        //закрываем ПЗК1
               "Control_PZK1".Avto_open := FALSE;
               "Control_PZK2".Mode := TRUE;        //закрываем ПЗК2
               "Control_PZK2".Avto_open := FALSE;
               "Control_KZ".Mode := TRUE;          //закрываем КЗ
               "Control_KZ".Avto_open := FALSE;
               "Control_KO".Mode := TRUE;          //закрываем КО
               "Control_KO".Avto_open := FALSE;
               "Control_KB".Mode := TRUE;          //открываем КБ
               "Control_KB".Avto_close := FALSE;
               "Control_IVN".Mode := TRUE;         //отключаем ИВН
               "Control_IVN".Avto_on := FALSE;
               "Control_ZDG".Mode := TRUE;         //закрываем ЗДГ
               "Control_ZDG".Avto_close := TRUE;
               "Control_ZDG".Avto_stop := FALSE;
               "Control_ZDG".Avto_open := FALSE;
               //запускаем контрольный таймер
               "Timer".VENTILATION_temp_PT := T#60s;
               "Timer".VENTILATION_temp_IN := TRUE;
               //проверяем положение ИМ по газу
               IF NOT "KB_close".Value AND //КБ открыт
                   NOT "KZ_open".Value AND //КЗ закрыт
                   NOT "KO_open".Value AND //КО закрыт
                   NOT "PZK1_open".Value AND   //ПЗК1 закрыт
                   NOT "PZK2_not_close".Value AND  //ПЗК2 закрыт
                   NOT "ZDG_no_close".Value THEN   //ЗДГ закрыт
                   //переход далее
                   "Timer".VENTILATION_temp_IN := FALSE;
                   "Message".VENTILATION_not_initial_state_gas := FALSE;
                   "Technology".Regim_ventilation_step := 2;
               END_IF;
               //если контрольное время вышло
               IF "Timer".VENTILATION_temp_Q THEN
                   "Message".VENTILATION_not_initial_state_gas := TRUE;
               END_IF;

           2:  //проверка нахождения ШУД ДС в дистаншионном режиме
               IF "DS_dist_control".Value THEN
                   //переход далее
                   "Message".VENTILATION_DS_need_dist_mode := FALSE;
                   "Technology".Regim_ventilation_step := 3;
               ELSE
                   "Message".VENTILATION_DS_need_dist_mode := TRUE;
               END_IF;

           3:  //проверка нахождения ШУД ДВ в дистаншионном режиме
               IF "DV_dist_control".Value THEN
                   //переход далее
                   "Message".VENTILATION_DV_need_dist_mode := FALSE;
                   "Technology".Regim_ventilation_step := 4;
               ELSE
                   "Message".VENTILATION_DV_need_dist_mode := TRUE;
               END_IF;

           4:  //проверка нахождения БРУ НАД в автоматическом режиме
               IF "NAD_avto".Value THEN
                   //переход далее
                   "Message".VENTILATION_BRU_NAD_need_avto_mode := FALSE;
                   "Technology".Regim_ventilation_step := 5;
               ELSE
                   "Message".VENTILATION_BRU_NAD_need_avto_mode := TRUE;
               END_IF;

           5:  //проверка нахождения БРУ НАВ в автоматическом режиме
               IF "NAV_avto".Value THEN
                   //переход далее
                   "Message".VENTILATION_BRU_NAV_need_avto_mode := FALSE;
                   "Technology".Regim_ventilation_step := 6;
               ELSE
                   "Message".VENTILATION_BRU_NAV_need_avto_mode := TRUE;
               END_IF;

           6:  //Закрытие НАД
               //Если ДС отключен, то
               IF NOT "DS_invertor_on".Value AND NOT "DS_powergrid_on".Value THEN
                   //закрываем НАД
                   "Control_NAD".Mode := TRUE;
                   "Control_NAD".Mode_from_PLC := FALSE;
                   "Control_NAD".Manual_close_from_PLC := TRUE;
                   "Control_NAD".SP_PID := 0.0;
                   //отключаем ДВ
                   "Control_DV".Mode := TRUE;
                   "Control_DV".Mode_from_PLC := FALSE;
                   "Control_DV".Avto_Stop := TRUE;
                   //закрываем НАВ
                   "Control_NAV".Mode := TRUE;
                   "Control_NAV".Mode_from_PLC := FALSE;
                   "Control_NAV".Manual_close_from_PLC := TRUE;
                   "Control_NAV".SP_PID := 0.0;
                   //контроль состояния НАД, ДВ, НАВ
                   IF "NAD_close".Value AND
                       (NOT "DV_invertor_on".Value AND NOT "DV_powergrid_on".Value) AND
                       "NAV_close".Value THEN
                       //переход далее
                       "Timer".VENTILATION_temp_IN := FALSE;
                       "Message".VENTILATION_not_initial_state_air := FALSE;
                       "Technology".Regim_ventilation_step := 7;
                   ELSE
                       //запускаем контрольный таймер
                       "Timer".VENTILATION_temp_PT := T#60s;
                       "Timer".VENTILATION_temp_IN := TRUE;
                   END_IF;
                   //если контрольное время вышло
                   IF "Timer".VENTILATION_temp_Q THEN
                       "Message".VENTILATION_not_initial_state_air := TRUE;
                       "Control_NAD".Manual_close_from_PLC := FALSE;
                       "Control_DV".Avto_Stop := FALSE;
                       "Control_NAV".Manual_close_from_PLC := FALSE;
                       //переходим в режим ОТКЛ на ожидание дальнейших действий
                       "Technology".Regim := 1;
                       "Technology".Regim_off_step := 1;
                   END_IF;
               ELSE
                   //переход далее
                   "Technology".Regim_ventilation_step := 7;
               END_IF;

           7:  //Закрытие НАВ
               //Если ДВ отключен, то
               IF NOT "DV_invertor_on".Value AND NOT "DV_powergrid_on".Value THEN
                   //закрываем НАВ
                   "Control_NAV".Mode := TRUE;
                   "Control_NAV".Mode_from_PLC := FALSE;
                   "Control_NAV".Manual_close_from_PLC := TRUE;
                   "Control_NAV".SP_PID := 0.0;
                   //контроль состояния НАВ
                   IF "NAV_close".Value THEN
                       //переход далее
                       "Timer".VENTILATION_temp_IN := FALSE;
                       "Message".VENTILATION_NAV_not_close := FALSE;
                       "Technology".Regim_ventilation_step := 8;
                   ELSE
                       //запускаем контрольный таймер
                       "Timer".VENTILATION_temp_PT := T#60s;
                       "Timer".VENTILATION_temp_IN := TRUE;
                   END_IF;
                   //если контрольное время вышло
                   IF "Timer".VENTILATION_temp_Q THEN
                       "Message".VENTILATION_NAV_not_close := TRUE;
                       "Control_NAV".Manual_close_from_PLC := FALSE;
                       //переходим в режим ОТКЛ на ожидание дальнейших действий
                       "Technology".Regim := 1;
                       "Technology".Regim_off_step := 1;
                   END_IF;
               ELSE
                   //переход далее
                   "Technology".Regim_ventilation_step := 8;
               END_IF;

           8:  //если ДС включен
               IF "DS_invertor_on".Value OR "DS_powergrid_on".Value THEN
                   //Взводим защиту Отключение ДС
                   "Alarm_Enable".DS_off := TRUE;
                   //переход на проверку состояния ДВ
                   "Technology".Regim_ventilation_step := 11;
               ELSE
                   //переход на включение ДС
                   "Technology".Regim_ventilation_step := 9;
               END_IF;

           9:  //пуск ДС
               "Control_DS".Mode := TRUE;
               IF NOT "Warning".DS_invertor_alarm THEN
                   "Control_DS".Avto_Start := TRUE;
               END_IF;
               "Control_DS".Mode_from_PLC := FALSE;
               //если выбран режим работы от ПЧ то задаем частоту 7Гц
               IF "DS_invertor_mode".Value THEN
                   "Control_DS".Manual_frequency_from_PLC := 7.0;
               ELSE
                   "Control_DS".Manual_frequency_from_PLC := 0.0;
               END_IF;
               //Проверяем включение ДС и отсутствие аварии ПЧ (в случае работы от ПЧ)
               IF ("DS_powergrid_mode".Value AND "DS_powergrid_on".Value) OR
                   ("DS_invertor_mode".Value AND "DS_invertor_on".Value AND NOT "Warning".DS_invertor_alarm) THEN
                   //Взводим защиту Отключение ДС
                   "Alarm_Enable".DS_off := TRUE;
                   //и переходим на задержку времени
                   "Timer".VENTILATION_temp_IN := FALSE;
                   "Message".VENTILATION_DS_not_on := FALSE;
                   "Technology".Regim_ventilation_step := 10;
               ELSE
                   //запускаем контрольный таймер
                   "Timer".VENTILATION_temp_PT := T#5s;
                   "Timer".VENTILATION_temp_IN := TRUE;
               END_IF;
               //если контрольное время вышло
               IF "Timer".VENTILATION_temp_Q THEN
                   "Message".VENTILATION_DS_not_on := TRUE;
               END_IF;

           10:  //задержка 6 сек
               "Timer".VENTILATION_temp_PT := T#6s;
               "Timer".VENTILATION_temp_IN := TRUE;
               //переход на проверку состояния ДВ
               IF "Timer".VENTILATION_temp_Q THEN
                   "Timer".VENTILATION_temp_IN := FALSE;
                   "Technology".Regim_ventilation_step := 11;
               END_IF;

           11:  //если ДВ включен
               IF "DV_invertor_on".Value OR "DV_powergrid_on".Value THEN
                   //Взводим защиту Отключение ДВ
                   "Alarm_Enable".DV_off := TRUE;
                   //переход на открытие НАД
                   "Technology".Regim_ventilation_step := 14;
               ELSE
                   //переход на включение ДВ
                   "Technology".Regim_ventilation_step := 12;
               END_IF;

           12: //пуск ДВ
               "Control_DV".Mode := TRUE;
               IF NOT "Warning".DV_invertor_alarm THEN
                   "Control_DV".Avto_Start := TRUE;
               END_IF;
               "Control_DV".Mode_from_PLC := FALSE;
               //если выбран режим работы от ПЧ то задаем частоту 7Гц
               IF "DV_invertor_mode".Value THEN
                   "Control_DV".Manual_frequency_from_PLC := 7.0;
               ELSE
                   "Control_DV".Manual_frequency_from_PLC := 0.0;
               END_IF;
               //Проверяем включение ДВ и отсутствие аварии ПЧ (в случае работы от ПЧ)
               IF ("DV_powergrid_mode".Value AND "DV_powergrid_on".Value) OR
                   ("DV_invertor_mode".Value AND "DV_invertor_on".Value AND NOT "Warning".DV_invertor_alarm) THEN
                   //Взводим защиту Отключение ДВ
                   "Alarm_Enable".DV_off := TRUE;
                   //и переходим на задержку времени
                   "Timer".VENTILATION_temp_IN := FALSE;
                   "Message".VENTILATION_DV_not_on := FALSE;
                   "Technology".Regim_ventilation_step := 13;
               ELSE
                   //запускаем контрольный таймер
                   "Timer".VENTILATION_temp_PT := T#5s;
                   "Timer".VENTILATION_temp_IN := TRUE;
               END_IF;
               //если контрольное время вышло
               IF "Timer".VENTILATION_temp_Q THEN
                   "Message".VENTILATION_DV_not_on := TRUE;
               END_IF;

           13: //задержка 6 сек
               "Timer".VENTILATION_temp_PT := T#6s;
               "Timer".VENTILATION_temp_IN := TRUE;
               //переход на открытие НАД
               IF "Timer".VENTILATION_temp_Q THEN
                   "Timer".VENTILATION_temp_IN := FALSE;
                   "Technology".Regim_ventilation_step := 14;
               END_IF;

           14: //НАД
               //Если ДС включен от ПЧ
               IF "DS_invertor_on".Value THEN
                   IF "NAD_open".Value THEN
                       "Technology".Regim_ventilation_step := 16;
                   ELSE
                       //полностью открываем НАД
                       "Control_NAD".Mode := TRUE;
                       "Control_NAD".Mode_from_PLC := FALSE;
                       "Control_NAD".Manual_open_from_PLC := TRUE;
                       IF NOT "NAD_avto".Value AND NOT "NAD_open".Value THEN
                           "Message".VENTILATION_NAD_not_open_manual := TRUE;
                       ELSE
                           "Message".VENTILATION_NAD_not_open_manual := FALSE;
                           "Technology".Regim_ventilation_step := 15;
                       END_IF;
                   END_IF;
               END_IF;
               //Если ДС включен от сети
               IF "DS_powergrid_on".Value THEN
                   //переводим ПИД НАД в автоматический режим на поддержание вентиляционных параметров
                   "Control_NAD".Mode := TRUE;
                   "Control_NAD".Mode_from_PLC := TRUE;
                   "Control_NAD".SP_PID := "RegMap".dP_furnace_ventilation;
                   //переход далее (на задержку времени)
                   "Timer".VENTILATION_temp_IN := FALSE;
                   "Technology".Regim_ventilation_step := 15;
               END_IF;

           15: //задержка 6 сек
               "Timer".VENTILATION_temp_PT := T#6s;
               "Timer".VENTILATION_temp_IN := TRUE;
               //переход на открытие НАВ
               IF "Timer".VENTILATION_temp_Q THEN
                   "Timer".VENTILATION_temp_IN := FALSE;
                   "Technology".Regim_ventilation_step := 16;
               END_IF;

           16: //НАВ
               //Если ДВ включен от ПЧ
               IF "DV_invertor_on".Value THEN
                   //полностью открываем НАВ
                   "Control_NAV".Mode := TRUE;
                   "Control_NAV".Mode_from_PLC := FALSE;
                   //контроль состояния НАВ
                   IF "NAV_open".Value THEN
                       "Control_NAV".Manual_open_from_PLC := FALSE;
                   ELSE
                       "Control_NAV".Manual_open_from_PLC := TRUE;
                   END_IF;
               END_IF;
               //Если ДВ включен от сети
               IF "DV_powergrid_on".Value THEN
                   //НАВ открываем до среднего положения
                   "Control_NAV".Mode := TRUE;
                   "Control_NAV".Mode_from_PLC := FALSE;
                   "Control_NAV".SP_PID := 0.0;
                   IF "NAV_middle".Value THEN
                       "Control_NAV".Manual_open_from_PLC := FALSE;
                   ELSE
                       "Control_NAV".Manual_open_from_PLC := TRUE;
                   END_IF;
               END_IF;

               IF NOT "NAV_avto".Value AND (("DV_invertor_on".Value AND NOT "NAV_open".Value) OR ("DV_powergrid_on".Value AND NOT "NAV_middle".Value)) THEN
                   "Message".VENTILATION_NAV_not_open_manual := TRUE;
               ELSE
                   "Message".VENTILATION_NAV_not_open_manual := FALSE;
               END_IF;

               IF (("DS_invertor_on".Value AND "NAD_open".Value) OR "DS_powergrid_on".Value) AND
                   (("DV_invertor_on".Value AND "NAV_open".Value) OR ("DV_powergrid_on".Value AND "NAV_middle".Value)) THEN
                   //переход далее
                   "Timer".VENTILATION_temp_IN := FALSE;
                   "Message".VENTILATION_NAV_or_NAD_not_open := FALSE;
                   "Technology".Regim_ventilation_step := 17;
               ELSE
                   //запускаем контрольный таймер
                   "Timer".VENTILATION_temp_PT := T#60s;
                   "Timer".VENTILATION_temp_IN := TRUE;
               END_IF;
               //если контрольное время вышло
               IF "Timer".VENTILATION_temp_Q THEN
                   "Message".VENTILATION_NAV_or_NAD_not_open := TRUE;
               END_IF;

           17: //задержка 1 сек
               "Timer".VENTILATION_temp_PT := T#1s;
               "Timer".VENTILATION_temp_IN := TRUE;
               //переход далее
               IF "Timer".VENTILATION_temp_Q THEN
                   "Timer".VENTILATION_temp_IN := FALSE;
                   "Technology".Regim_ventilation_step := 18;
               END_IF;

           18: //включаем ПИД ДС (если режим работы от ПЧ)
               IF "DS_invertor_mode".Value THEN
                   IF "Control_DS".Mode = TRUE AND
                       "Control_DS".Mode_from_PLC = TRUE AND
                       "Control_DS".SP_PID = "RegMap".dP_furnace_ventilation THEN
                       "Timer".VENTILATION_temp_IN := FALSE;
                       "Technology".Regim_ventilation_step := 20;
                   ELSE
                       "Control_DS".Mode := TRUE;
                       "Control_DS".Mode_from_PLC := TRUE;
                       "Control_DS".SP_PID := "RegMap".dP_furnace_ventilation;
                       //переход на следующий шаг
                       "Timer".VENTILATION_temp_IN := FALSE;
                       "Technology".Regim_ventilation_step := 19;
                   END_IF;
               ELSE
                   "Control_DS".Mode_from_PLC := FALSE;
                   //переход через шаг (без ожидания)
                   "Timer".VENTILATION_temp_IN := FALSE;
                   "Technology".Regim_ventilation_step := 20;
               END_IF;

           19: //Ожидаем 6 сек
               "Timer".VENTILATION_temp_PT := T#6s;
               "Timer".VENTILATION_temp_IN := TRUE;
               //переход на следующий шаг
               IF "Timer".VENTILATION_temp_Q THEN
                   "Timer".VENTILATION_temp_IN := FALSE;
                   "Technology".Regim_ventilation_step := 20;
               END_IF;

